(* IEC 61131-3 sources: SmartHomeNew/ (part 16) *)

(* ---- PRG_System.st ---- *)
PROGRAM PRG_System
VAR

// === SENSOR PROCESSING (SHADOW) ===
fbSensorCO : FB_Sensor_Analog_Processing;
fbCalibCO  : FB_Sensor_Calibration_Processor;
fbSensorMethane : FB_Sensor_Analog_Processing;
fbCalibMethane  : FB_Sensor_Calibration_Processor;
fbSmokeDetector : FB_Smoke_Detector;
L_CO_Processed : REAL;
L_CO_Calibrated : REAL;
L_Safety_Selector_i : INT;
L_Methane_Processed : REAL;
L_Methane_Calibrated : REAL;
L_Smoke_Detected : BOOL;

// === LIFETIME MANAGERS ===
fbLifetimePump : FB_Lifetime_Manager;
fbLifetimeFan  : FB_Lifetime_Manager;

    // === TREND WRITE CONTROL ===
    L_Trend_Write : BOOL;
    L_Trend_Write_Prev : BOOL;

    // === TREND → HISTORY BRIDGE ===
    L_Trend_Event : ST_History_Record;

    // === TREND SYSTEM (MVP) ===
    L_Trend_Logger : FB_Trend_Logger;
    L_Trend_Data : ST_Trend_Data;
    L_Trend_Adapter : FB_Trend_Adapter;
    L_Trend_Avg : REAL;
    L_Trend_Min : REAL;
    L_Trend_Max : REAL;
    L_Trend_Up : BOOL;
    L_Trend_Down : BOOL;
    L_Trend_Last_Write_MS : UDINT;
    L_Trend_Last_Written_Avg : REAL;
    L_Trend_Write_Allowed : BOOL;
    L_i : INT;
    L_Motion_Sensors_16 : ARRAY[1..16] OF BOOL;
    // --- ADAPTER LAYER ---
    L_Zone_Valves_8 : ARRAY[1..8] OF BOOL;
    L_Lighting_32   : ARRAY[1..32] OF BYTE;
    L_Lighting_Bool_32 : ARRAY[1..32] OF BOOL;
    L_FloorTemps_8  : ARRAY[1..8] OF REAL;
    fbCoreKernelObserver : FB_CoreKernel_Live_Observer;
    fbSystemHealth : FB_System_Health;
    fbRedundancy : FB_Redundancy_Manager;
    fbGateway : FB_Gateway_Interface;
    fbScenarioManager : FB_Scenario_Manager;
    fbScenarioGuard : FB_Scenario_Transition_Guard;
    fbSimulationManager : FB_Simulation_Manager;
    fbRuleEngine : FB_Rule_Engine;
    fbNVRAMManager : FB_NVRAM_Manager;

    fbBlackBox : FB_BlackBox_Recorder;
    fbAstroTimer : FB_Astro_Timer;
    fbAlarmManager : FB_Alarm_Manager;
    fbHistoryManager : FB_History_Manager;
    fbSafety : FB_Safety_Manager;
    fbStateManager : FB_State_Manager;
    fbWatchdog : FB_Watchdog;
    fbHMIInterface : FB_HMI_Interface;
    fbFaultLogger : FB_Fault_Logger;
    fbLogEvent : FB_LogEvent;

    L_Time_Diff : UDINT;
    L_Local_State : ST_System_State_Snapshot;
    L_Remote_State : ST_System_State_Snapshot;
    L_NVRAM_Cmd : BYTE;
    L_NVRAM_Offset : UDINT;
    L_NVRAM_Done : BOOL;
    L_NVRAM_Err : BOOL;
    L_NVRAM_ErrID : UDINT;
    L_BB_Record : ST_BlackBox_Record;
    L_BB_Freeze : BOOL;
    L_Scenario_Idx : INT;
        L_Last_Operator_Blocked : BOOL;
    L_Last_DHW_Heating_In_Service : BOOL;
    L_Last_DHW_Circ_In_Service : BOOL;
    L_Dangerous_Action_Armed : BOOL;
    L_Dangerous_Action_Deadline_MS : UDINT;
    L_Maintenance_Apply_Intent : BOOL;
    L_Last_System_Mode : E_System_Operating_Mode;
    L_Last_First_Fault_Type : INT;
    L_Last_First_Fault_Source : INT;
    L_Last_Root_Cause : E_System_Root_Cause;
    L_History_Event : ST_History_Record;
    L_History_Write_Event : BOOL;
    L_Last_Operator_Journal_Seq : UDINT;
    L_Last_Maintenance_Action_Code : UDINT;
    L_Last_Event_Code : UDINT;
    L_Last_Event_Value : REAL;
    L_Last_Event_Time_MS : UDINT;
    L_Gateway_Writes_Allowed : BOOL;
    L_Last_Policy_Event_Time_MS : UDINT;

    L_Scenario_Req_Operator : E_SCENARIO_TYPE;
    L_Scenario_Req_Gateway  : E_SCENARIO_TYPE;
    L_Scenario_Req_Rule     : E_SCENARIO_TYPE;
    L_Scenario_Req_Final    : E_SCENARIO_TYPE; // TRACE ONLY: arbitration result before policy
    L_Scenario_Intent       : E_SCENARIO_TYPE;
L_Scenario_Source       : E_SCENARIO_SOURCE;

L_IO_Fault_Prev : BOOL;
L_Watchdog_Fault_Prev : BOOL;
L_Comm_Fault_Prev : BOOL;
L_Sensor_Fault_Prev : BOOL;
L_Subsystem_Fault_Prev : BOOL;
L_Mode_Prev : E_System_Operating_Mode;
L_User_Access_Denied_Prev : BOOL;
L_Dangerous_Action_Request_Prev : BOOL;

    L_Persist_Buffer : ARRAY[0..4] OF BYTE;
    L_Last_Written_Persist_Buffer : ARRAY[0..4] OF BYTE;
    L_Persist_Buffer_Changed : BOOL;
    L_Last_Persist_Write_MS : UDINT;
    L_Recovery_Done : BOOL;
    L_Persist_Struct : ST_Persist;
END_VAR

// 0. Инициализация RETAIN переменных при первом запуске
IF NOT GVL_Retain.G_Initialized THEN
    FOR L_i := 0 TO GVL_CONSTANTS.C_MAX_PRESENCE_HISTORY - 1 DO
        GVL_Retain.G_Presence_History[L_i] := 0;
    END_FOR;

    GVL_Retain.G_History_Write_Idx := 1;
    GVL_Retain.G_History_Total_Events := 0;

    FOR L_i := 1 TO GVL_CONSTANTS.C_MAX_BOILERS DO
        GVL_Retain.G_Boiler_Accumulated_MS[L_i] := 0;
        GVL_Retain.G_Boiler_Work_Seconds[L_i] := 0;
    END_FOR;

    FOR L_i := 1 TO GVL_CONSTANTS.C_MAX_MANIFOLDS DO
        GVL_Retain.G_Valve_Test_Results[L_i] := FALSE;
    END_FOR;

    L_Local_State.Version := 0;
    L_Remote_State.Version := 0;

    GVL_Retain.G_Initialized := TRUE;

END_IF;

// === NVRAM RECOVERY (ONCE AFTER BOOT) ===
IF NOT L_Recovery_Done THEN
    IF GVL_PERSISTENT.P_Valid THEN
        GVL_STATE.G_Safety_Gas_Latched := GVL_PERSISTENT.P_Safety_Gas_Latched;
        GVL_STATE.G_Safety_Smoke_Latched := GVL_PERSISTENT.P_Safety_Smoke_Latched;
        GVL_STATE.G_Safety_Leak_Latched := GVL_PERSISTENT.P_Safety_Leak_Latched;
        GVL_STATE.G_System_Mode := GVL_PERSISTENT.P_System_Mode;
    END_IF;

    L_Recovery_Done := TRUE;
END_IF;

// NVRAM CONTROLLED WRITE ENABLED (step 8B)

// 1. Обновление системного времени
GVL_STATUS.G_System_Time_MS := TIME_TO_UDINT(TIME());
L_Time_Diff := (SEL(GVL_STATUS.G_System_Time_MS >= GVL_STATUS.G_Last_System_Time_MS, GVL_STATUS.G_System_Time_MS - GVL_STATUS.G_Last_System_Time_MS, (4294967295 - GVL_STATUS.G_Last_System_Time_MS) + GVL_STATUS.G_System_Time_MS + 1));
GVL_STATUS.G_Time_Of_Day_MS := (GVL_STATUS.G_Time_Of_Day_MS + L_Time_Diff) MOD 86400000;

IF GVL_STATUS.G_Time_Of_Day_MS < L_Time_Diff THEN
    GVL_STATUS.G_Current_Day := (GVL_STATUS.G_Current_Day MOD 7) + 1;
    GVL_STATUS.G_Day_Of_Year := (GVL_STATUS.G_Day_Of_Year MOD 365) + 1;
END_IF;

GVL_STATUS.G_Last_System_Time_MS := GVL_STATUS.G_System_Time_MS;
GVL_STATUS.G_Current_TOD := UDINT_TO_TOD(GVL_STATUS.G_Time_Of_Day_MS);

// Формирование локального состояния для репликации
L_Local_State.System_Time_MS := GVL_STATUS.G_System_Time_MS;
L_Local_State.Current_Scenario := GVL_STATUS.G_Current_Scenario;
L_Local_State.Security_Armed := GVL_ALARM.G_Security_Armed;
L_Local_State.Active_Alarms := GVL_ALARM.G_Active_Alarm_Count;
L_Local_State.Zone_Valves := GVL_STATE.G_Zone_Valves;
L_Local_State.Manifold_Pumps := GVL_STATE.G_Manifold_Pumps;
L_Local_State.Lighting_States := GVL_STATE.G_Lighting_Levels;
L_Local_State.Blinds_Positions := GVL_STATE.G_Blinds_Positions;
L_Local_State.Socket_States := GVL_STATE.G_Socket_States;
L_Local_State.Gas_Valve_Closed := GVL_COMMAND.G_Gas_Valve_Close;
L_Local_State.Water_Valves_Closed := GVL_COMMAND.G_Close_Valve_36;
L_Local_State.Version := L_Local_State.Version + 1;

// 2. Определение роли ПЛК (Active/Standby)
fbRedundancy(
    VI_System_Time_MS := GVL_STATUS.G_System_Time_MS,
    VI_Local_PLC_ID := GVL_STATUS.G_PLC_ID,
    VI_Remote_Pulse := GVL_IO.DI_Partner_Pulse,
    VI_Remote_Is_Active := GVL_IO.DI_Partner_Active,
    VI_Gateway_Ping_OK := GVL_GATEWAY.G_Gateway_Ping_OK,
    VI_Local_State := L_Local_State,
    VI_Remote_State := L_Remote_State
);
GVL_STATUS.G_Is_Active_PLC := (fbRedundancy.VO_Local_Role = E_PLC_ROLE.ROLE_ACTIVE);
GVL_IO.DO_Heartbeat_Pulse := fbRedundancy.VO_Local_Pulse;
GVL_IO.DO_Active_Status := GVL_STATUS.G_Is_Active_PLC;

// 3. Синхронизация состояния (применение полученного состояния)
IF fbRedundancy.VO_State_Updated THEN
    GVL_STATUS.G_Current_Scenario := fbRedundancy.VO_Synced_State.Current_Scenario;
    GVL_ALARM.G_Security_Armed := fbRedundancy.VO_Synced_State.Security_Armed;
    GVL_STATE.G_Zone_Valves := fbRedundancy.VO_Synced_State.Zone_Valves;
    GVL_STATE.G_Manifold_Pumps := fbRedundancy.VO_Synced_State.Manifold_Pumps;
    GVL_STATE.G_Lighting_Levels := fbRedundancy.VO_Synced_State.Lighting_States;
    GVL_STATE.G_Blinds_Positions := fbRedundancy.VO_Synced_State.Blinds_Positions;
    GVL_STATE.G_Socket_States := fbRedundancy.VO_Synced_State.Socket_States;
    GVL_COMMAND.G_Gas_Valve_Close := fbRedundancy.VO_Synced_State.Gas_Valve_Closed;
    GVL_COMMAND.G_Close_Valve_36 := fbRedundancy.VO_Synced_State.Water_Valves_Closed;
    L_Local_State.Version := fbRedundancy.VO_Synced_State.Version;
END_IF;

fbSafety(
    VI_Gas_Alarm := GVL_STATE.G_Safety_Gas_Alarm,
    VI_Leak_Alarm := GVL_STATE.G_Safety_Leak_Alarm,
    VI_Smoke_Alarm := GVL_STATE.G_Safety_Smoke_Alarm,
    VI_Reset := GVL_COMMAND.G_Reset_Errors,
    VO_Gas_Latched => GVL_STATE.G_Safety_Gas_Latched,
    VO_Leak_Latched => GVL_STATE.G_Safety_Leak_Latched,
    VO_Smoke_Latched => GVL_STATE.G_Safety_Smoke_Latched,
    VO_Emergency_Stop => GVL_STATE.G_Safety_Emergency_Stop
);

// 3.4. Агрегация состояния anti-freeze hardware
GVL_STATE.G_Freeze_Hardware_Degraded := GVL_STATUS.G_Diagnostics.Backup_Pump_Fault OR GVL_STATUS.G_Diagnostics.Electric_Heater_Fault;
GVL_STATE.G_Freeze_Hardware_Failed := GVL_STATUS.G_Diagnostics.Backup_Pump_Fault AND GVL_STATUS.G_Diagnostics.Electric_Heater_Fault;

// 3.6. Health manager: новая интеграция safety + diagnostics + watchdog
fbWatchdog(
    VI_System_Time_MS := GVL_STATUS.G_System_Time_MS
);

fbSystemHealth(
    VI_Smoke_Detected := GVL_HEALTH_BRIDGE.G_Smoke_Detected OR GVL_STATE.G_Safety_Smoke_Latched,
    VI_Gas_Detected := GVL_HEALTH_BRIDGE.G_Gas_Detected OR GVL_STATE.G_Safety_Gas_Latched,
    VI_CO_Warning_Level := GVL_HEALTH_BRIDGE.G_CO_Warning_Level,
    VI_CO_Alarm_Level := GVL_HEALTH_BRIDGE.G_CO_Alarm_Level,
    VI_Leak_Detected := GVL_HEALTH_BRIDGE.G_Leak_Detected OR GVL_STATE.G_Safety_Leak_Latched,
    VI_Sensor_Fault := GVL_STATE.G_Heating_Sensor_Fault OR GVL_STATE.G_DHW_Sensor_Fault,
    VI_IO_Offline := GVL_STATE.G_Heating_IO_Fault OR GVL_STATE.G_DHW_IO_Fault OR GVL_STATE.G_Ventilation_IO_Fault OR GVL_STATE.G_Lighting_IO_Fault,
    VI_Comm_Fault := GVL_STATE.G_Access_Comm_Fault,
    VI_Watchdog_Fault := fbWatchdog.VO_Watchdog_Fault,
    VI_Subsystem_Fault := GVL_STATE.G_Heating_Subsystem_Degraded OR GVL_STATE.G_DHW_Subsystem_Degraded OR GVL_STATE.G_Ventilation_Subsystem_Degraded
);

// 3.6. State manager: агрегированная логика режима работы
fbStateManager(
    VI_System_Severity := fbSystemHealth.VO_System_Severity,
    VI_Root_Cause := fbSystemHealth.VO_Root_Cause,
    VI_Freeze_Risk := GVL_STATE.G_Safety_Freeze_Risk
);

fbHMIInterface(
    VI_Severity := fbSystemHealth.VO_System_Severity,
    VI_RootCause := fbSystemHealth.VO_Root_Cause,
    VI_Status_Msg := fbStateManager.VO_Status_Msg
);

fbFaultLogger(
    VI_Severity := fbSystemHealth.VO_System_Severity,
    VI_RootCause := fbSystemHealth.VO_Root_Cause,
    VI_Time_MS := GVL_STATUS.G_System_Time_MS
);

// publish integrated outputs
GVL_STATUS.G_System_Mode_Msg := fbStateManager.VO_Status_Msg;

// === DIAGNOSTIC FLAGS (export) ===
GVL_STATUS.G_Diagnostics.Sensor_Fault :=
    GVL_STATE.G_Heating_Sensor_Fault OR
    GVL_STATE.G_DHW_Sensor_Fault;

GVL_STATUS.G_Diagnostics.IO_Offline :=
    GVL_STATE.G_Heating_IO_Fault OR
    GVL_STATE.G_DHW_IO_Fault OR
    GVL_STATE.G_Ventilation_IO_Fault OR
    GVL_STATE.G_Lighting_IO_Fault;

GVL_STATUS.G_Diagnostics.Subsystem_Degraded :=
    GVL_STATE.G_Heating_Subsystem_Degraded OR
    GVL_STATE.G_DHW_Subsystem_Degraded OR
    GVL_STATE.G_Ventilation_Subsystem_Degraded;

GVL_GATEWAY.G_Gateway_HMI_Status_Message := fbHMIInterface.VO_HMI_Status_Text;
IF fbFaultLogger.VO_Last_Event_Text <> '' THEN
    GVL_HEALTH_BRIDGE.G_Last_Fault_Event_Text := fbFaultLogger.VO_Last_Event_Text;
END_IF;

// 3.7. Применение вычисленного режима системы
GVL_STATE.G_System_Mode := fbStateManager.VO_System_Mode;

CASE GVL_STATE.G_System_Mode OF
    E_System_Operating_Mode.MODE_SAFE_STOP:
        GVL_STATE.G_System_Mode_Text := 'SAFE_STOP';

    E_System_Operating_Mode.MODE_FREEZE_PROTECTION:
        GVL_STATE.G_System_Mode_Text := 'FREEZE_PROTECTION';

    E_System_Operating_Mode.MODE_DEGRADED:
        GVL_STATE.G_System_Mode_Text := 'DEGRADED';

    ELSE
        GVL_STATE.G_System_Mode_Text := 'NORMAL';
END_CASE;

CASE fbSystemHealth.VO_Root_Cause OF
    E_System_Root_Cause.ROOT_FIRE:
        GVL_STATUS.G_System_Mode_Cause := 'Пожар/дым';
    E_System_Root_Cause.ROOT_GAS_LEAK:
        GVL_STATUS.G_System_Mode_Cause := 'Утечка газа';
    E_System_Root_Cause.ROOT_CO_CRITICAL:
        GVL_STATUS.G_System_Mode_Cause := 'Критический CO';
    E_System_Root_Cause.ROOT_CO_WARNING:
        GVL_STATUS.G_System_Mode_Cause := 'Повышенный CO';
    E_System_Root_Cause.ROOT_WATER_LEAK:
        GVL_STATUS.G_System_Mode_Cause := 'Протечка воды';
    E_System_Root_Cause.ROOT_WATCHDOG_FAULT:
        GVL_STATUS.G_System_Mode_Cause := 'Ошибка watchdog';
    E_System_Root_Cause.ROOT_IO_OFFLINE:
        GVL_STATUS.G_System_Mode_Cause := 'Недоступен модуль IO';
    E_System_Root_Cause.ROOT_COMM_FAULT:
        GVL_STATUS.G_System_Mode_Cause := 'Ошибка связи';
    E_System_Root_Cause.ROOT_SENSOR_FAULT:
        GVL_STATUS.G_System_Mode_Cause := 'Ошибка датчика';
    E_System_Root_Cause.ROOT_SUBSYSTEM_FAULT:
        GVL_STATUS.G_System_Mode_Cause := 'Ошибка подсистемы';
    ELSE
        GVL_STATUS.G_System_Mode_Cause := 'Аварийные режимы отсутствуют';
END_CASE;

// final status text comes from State_Manager
GVL_STATUS.G_System_Mode_Msg := fbStateManager.VO_Status_Msg;

// 3.6a. Расчёт направленной эвакуации
FOR L_i := 1 TO 32 DO
    GVL_STATE.G_Evac_Guidance[L_i] := 0;

    IF GVL_STATE.G_Evac_Hazard_Zone[L_i] THEN
        GVL_STATE.G_Evac_Guidance[L_i] := -1;
    END_IF;

    IF GVL_CONFIG.G_Evac_Exit_Zones[L_i] AND NOT GVL_STATE.G_Evac_Hazard_Zone[L_i] THEN
        GVL_STATE.G_Evac_Guidance[L_i] := 1;
    END_IF;
END_FOR;

// 3.5a. Вычисление человекочитаемых имён зон эвакуации для HMI
GVL_STATUS.G_Evac_Target_Zone_Name := '';
GVL_STATUS.G_Evac_Hazard_Zone_Name := '';

FOR L_i := 1 TO 32 DO
    IF (GVL_STATUS.G_Evac_Hazard_Zone_Name = '') AND GVL_STATE.G_Evac_Hazard_Zone[L_i] THEN
        GVL_STATUS.G_Evac_Hazard_Zone_Name := GVL_CONFIG.G_Evac_Zone_Names[L_i];
        IF GVL_STATUS.G_Evac_Hazard_Zone_Name = '' THEN
            GVL_STATUS.G_Evac_Hazard_Zone_Name := CONCAT('Zone ', INT_TO_STRING(L_i));
        END_IF;
    END_IF;

    IF (GVL_STATUS.G_Evac_Target_Zone_Name = '') AND (GVL_STATE.G_Evac_Guidance[L_i] = 1) THEN
        GVL_STATUS.G_Evac_Target_Zone_Name := GVL_CONFIG.G_Evac_Zone_Names[L_i];
        IF GVL_STATUS.G_Evac_Target_Zone_Name = '' THEN
            GVL_STATUS.G_Evac_Target_Zone_Name := CONCAT('Zone ', INT_TO_STRING(L_i));
        END_IF;
    END_IF;
END_FOR;

// 3.6. Активация световой эвакуации
IF GVL_STATE.G_System_Mode = E_System_Operating_Mode.MODE_SAFE_STOP AND GVL_STATE.G_Safety_Smoke_Latched THEN
    GVL_STATE.G_Evacuation_Lighting_Active := TRUE;
ELSE
    GVL_STATE.G_Evacuation_Lighting_Active := FALSE;
END_IF;

// 4. Астрономический таймер
fbAstroTimer(
    VI_System_Time_MS := GVL_STATUS.G_System_Time_MS,
    VI_Latitude := 55.75,
    VI_Longitude := 37.61,
    VI_Day_Of_Year := GVL_STATUS.G_Day_Of_Year,
    VO_Is_Night => GVL_STATUS.G_Is_Night
);

// 5. Управление сценариями
// Scenario request (direct + early operator gate)
IF GVL_STATE.G_System_Mode = E_System_Operating_Mode.MODE_NORMAL THEN
    L_Scenario_Req_Operator := GVL_COMMAND.G_Scenario_Request_Operator;
ELSE
    L_Scenario_Req_Operator := E_SCENARIO_TYPE.SCENARIO_NONE;
END_IF;
L_Scenario_Req_Gateway := 0;
L_Scenario_Req_Rule := 0;

// Синхронизируем request с фактически активным сценарием

L_Scenario_Idx := TO_INT(GVL_STATUS.G_Current_Scenario);
IF L_Scenario_Idx < 0 OR L_Scenario_Idx > 7 THEN
    L_Scenario_Idx := 0;
END_IF;

// 6. Симуляция присутствия
fbSimulationManager(
    VI_System_Time_MS := GVL_STATUS.G_System_Time_MS,
    VI_IsActivePLC := GVL_STATUS.G_Is_Active_PLC AND (GVL_STATE.G_System_Mode = E_System_Operating_Mode.MODE_NORMAL),
    VI_Scenario := GVL_STATUS.G_Current_Scenario,
    VI_Config := GVL_CONFIG.G_HMI_Scenario_Configs[L_Scenario_Idx],
    VO_Sim_Lights => GVL_STATE.G_Sim_Lights,
    VO_Sim_Active => GVL_STATUS.G_Sim_Active
);

// 6.5. Пользовательские правила (Rule Engine)
fbRuleEngine(
    VI_System_Time_MS := GVL_STATUS.G_System_Time_MS,
    VI_IsActivePLC := GVL_STATUS.G_Is_Active_PLC,
    VI_Rules := GVL_CONFIG.G_HMI_User_Rules,
    VI_Indoor_Temps := GVL_STATE.G_Room_Temps,
    VI_Floor_Temps := L_FloorTemps_8,
    VI_Humidities := GVL_STATE.G_Room_Hum,
    VI_CO2_Levels := GVL_STATE.G_Room_CO2,
    VI_Motion_Sensors := L_Motion_Sensors_16,
    VI_Door_Sensors := GVL_STATE.G_Door_Sensors,
    VI_Window_Sensors := GVL_STATE.G_Window_Sensors,
    VI_Water_Sensors := GVL_STATE.G_Water_Sensors,
    VI_Smoke_Sensors := GVL_STATE.G_Smoke_Sensors,
    VI_Methane_Sensors := GVL_STATE.G_Methane_Sensors,
    VI_CO_Sensors := GVL_STATE.G_CO_Sensors,
    VI_Security_Armed := GVL_ALARM.G_Security_Armed,
    VI_Current_Time := GVL_STATUS.G_Current_TOD,
    VI_Day_Of_Week := TO_INT(GVL_STATUS.G_Current_Day),
    VO_Actions => GVL_STATE.G_Rule_Actions
);

FOR L_i := 1 TO GVL_CONSTANTS.C_MAX_RULES DO
    IF GVL_STATE.G_Rule_Actions[L_i].Active AND GVL_STATE.G_Rule_Actions[L_i].Action_Type = E_Rule_Action_Type.ACTION_ACTIVATE_SCENARIO THEN
        L_Scenario_Req_Rule := TO_BYTE(GVL_STATE.G_Rule_Actions[L_i].Value);
    END_IF;
END_FOR;

// 8.5 Менеджер тревог (Сбор всех аварий)
fbAlarmManager(
    VI_System_Time_MS := GVL_STATUS.G_System_Time_MS,
    VI_IsActivePLC := GVL_STATUS.G_Is_Active_PLC,
    VI_Gas_Alarm := GVL_ALARM.G_Gas_Alarm_Active,
    VI_Fire_Alarm := GVL_ALARM.G_Fire_Alarm_Active,
    VI_Flood_Alarm := GVL_ALARM.G_Flood_Alarm_Active,
    VI_Security_Alarm := GVL_ALARM.G_Security_Alarm,
    VI_First_Fault_Active := fbSystemHealth.VO_First_Fault_Active,
    VI_First_Fault_Type := fbSystemHealth.VO_First_Fault_Type,
    VI_First_Fault_Source := fbSystemHealth.VO_First_Fault_Source,
    VI_Boiler_Errors := GVL_STATE.G_Boiler_Error,
    VI_Security_Msg := GVL_STATUS.G_Security_Status_Msg,
    VI_Acknowledge_All := GVL_CONFIG.G_HMI_Ack_Alarms OR GVL_COMMAND.G_Reset_Errors,
    VI_Mute_Siren := GVL_CONFIG.G_HMI_Mute_Alarm,
    VIO_Next_Alarm_ID := GVL_ALARM.G_Next_Alarm_ID,
    VO_Global_Critical => GVL_ALARM.G_Global_Critical,
    VO_Global_Warning => GVL_ALARM.G_Global_Warning,
    VO_Siren_Active => GVL_ALARM.G_Global_Siren,
    VO_Active_Count => GVL_ALARM.G_Active_Alarm_Count,
    VO_Unacked_Count => GVL_ALARM.G_Unacked_Alarm_Count,
    VO_Event_Pulse => GVL_STATUS.G_Diagnostics.Alarm_Event_Pulse,
    VO_Event_Code => GVL_STATUS.G_Diagnostics.Alarm_Event_Code,
    VO_Event_Value => GVL_STATUS.G_Diagnostics.Alarm_Event_Value,
    VO_Alarm_List => GVL_ALARM.G_Alarm_List
);

// Command arbitration: OPERATOR > GATEWAY
L_Gateway_Writes_Allowed :=
    NOT GVL_STATUS.G_Diagnostics.Dangerous_Action_Pending_Confirm AND
    NOT GVL_STATUS.G_Diagnostics.Operator_Action_Blocked AND
    NOT GVL_STATUS.G_Diagnostics.User_Access_Denied;

// 13. Интерфейс шлюза (Modbus TCP)
fbGateway(
    VI_System_Time_MS := GVL_STATUS.G_System_Time_MS,
    VI_Local_PLC_Role := SEL(GVL_STATUS.G_Is_Active_PLC, E_PLC_ROLE.ROLE_STANDBY, E_PLC_ROLE.ROLE_ACTIVE),
    VI_Incoming_Command := GVL_GATEWAY.G_Gateway_Command,
    VI_Command_Received := GVL_GATEWAY.G_Gateway_Command_Received,
    VI_FloorHeating_Temps := L_FloorTemps_8,
    VI_Room_Temps := GVL_STATE.G_Room_Temps,
    VI_Zone_Valve_States := L_Zone_Valves_8,
    VI_Manifold_Pressures := GVL_STATE.G_Manifold_Pressures,
    VI_Manifold_Pump_States := GVL_STATE.G_Manifold_Pumps,
    VI_Outdoor_Temp := GVL_STATE.G_Outdoor_Temp,
    VI_Security_Armed := GVL_ALARM.G_Security_Armed,
    VI_Flood_Alarm_Active := GVL_ALARM.G_Flood_Alarm_Active,
    VI_Gas_Alarm_Active := GVL_ALARM.G_Gas_Alarm_Active,
    VI_Fire_Alarm_Active := GVL_ALARM.G_Fire_Alarm_Active,
    VI_Methane_Concentration := GVL_STATE.G_Methane_Sensors[1],
    VI_Lighting_Base_Levels := L_Lighting_32,
    VI_Socket_States := GVL_STATE.G_Socket_States,
    VI_Blinds_Positions := GVL_STATE.G_Blinds_Positions,
    VI_Active_Scenario := GVL_STATUS.G_Current_Scenario,
    VI_Send_2FA_Req := GVL_COMMAND.G_Send_2FA_Req,
    VI_2FA_Code := GVL_COMMAND.G_2FA_Code_Out,
    VI_Allowed_IPs := GVL_CONFIG.G_Allowed_IPs,
    VO_Telegram_Msg => GVL_GATEWAY.G_Gateway_Telegram_Msg,
    VO_Send_Telegram => GVL_GATEWAY.G_Gateway_Send_Telegram,
    VO_HMI_Status_Message => GVL_GATEWAY.G_Gateway_HMI_Status_Message,

    VO_Data_Ready => GVL_GATEWAY.G_Gateway_Data_Ready,
    VO_Modbus_Registers => GVL_GATEWAY.G_Gateway_Modbus_Registers,
    VO_Arm_Req => GVL_COMMAND.G_Arm_Req,
    VO_Disarm_Req => GVL_COMMAND.G_Disarm_Req,
    VO_PIN_Code => GVL_COMMAND.G_PIN_Code,
    VO_RFID_Tag => GVL_COMMAND.G_RFID_Tag,
    VO_2FA_Code_In => GVL_COMMAND.G_2FA_Code_In,
    VO_Lighting_Override => GVL_COMMAND.G_Lighting_Override,
    VO_Blinds_Override => GVL_COMMAND.G_Blinds_Override,
    VO_Socket_Override => GVL_COMMAND.G_Socket_Override,
    VO_Reset_Errors_Req => GVL_COMMAND.G_Reset_Errors
);

IF L_Gateway_Writes_Allowed AND
   fbGateway.VO_Set_Scenario_Req AND
   ((GVL_STATE.G_System_Mode = E_System_Operating_Mode.MODE_NORMAL) OR
    (GVL_STATE.G_System_Mode = E_System_Operating_Mode.MODE_DEGRADED)) THEN
    L_Scenario_Req_Gateway := fbGateway.VO_Target_Scenario;
END_IF;

IF L_Gateway_Writes_Allowed AND
   fbGateway.VO_Set_Temp_Req AND
   (GVL_STATE.G_System_Mode = E_System_Operating_Mode.MODE_NORMAL) THEN
    GVL_CONFIG.G_HMI_FloorHeating_Configs[fbGateway.VO_Target_Zone].design_temp := fbGateway.VO_Target_Temp;
END_IF;

IF L_Gateway_Writes_Allowed AND
   fbGateway.VO_Set_Vent_Req AND
   (GVL_STATE.G_System_Mode = E_System_Operating_Mode.MODE_NORMAL) THEN
    GVL_CONFIG.G_HMI_Vent_Global_Config.default_supply_speed := fbGateway.VO_Target_Vent_Speed;
END_IF;

IF L_Gateway_Writes_Allowed AND
   fbGateway.VO_Set_Config_Req AND
   (GVL_STATE.G_System_Mode = E_System_Operating_Mode.MODE_NORMAL) THEN
    GVL_CONFIG.G_HMI_Apply_Settings := TRUE;
END_IF;

IF L_Gateway_Writes_Allowed AND
   fbGateway.VO_Sync_Time_Req AND
   (GVL_STATE.G_System_Mode = E_System_Operating_Mode.MODE_NORMAL) THEN
    GVL_STATUS.G_Time_Of_Day_MS := fbGateway.VO_New_Time_MS;
END_IF;

// === SCENARIO REQUEST VALIDATION ===
// Normalize invalid values to NONE to avoid corrupt inputs.
// Actual enum range in E_SCENARIO_TYPE is 0..7.
IF TO_USINT(L_Scenario_Req_Operator) > 7 THEN
    L_Scenario_Req_Operator := E_SCENARIO_TYPE.SCENARIO_NONE;
END_IF;

IF TO_USINT(L_Scenario_Req_Gateway) > 7 THEN
    L_Scenario_Req_Gateway := E_SCENARIO_TYPE.SCENARIO_NONE;
END_IF;

IF TO_USINT(L_Scenario_Req_Rule) > 7 THEN
    L_Scenario_Req_Rule := E_SCENARIO_TYPE.SCENARIO_NONE;
END_IF;

// ================= COMMAND GATE (FINAL) =================
IF GVL_STATE.G_System_Mode = E_System_Operating_Mode.MODE_SAFE_STOP THEN

    // Блокируем ВСЕ опасные команды после Gateway
    GVL_COMMAND.G_Scenario_Request_Operator := 0;

    FOR L_i := 1 TO 32 DO
        GVL_COMMAND.G_Lighting_Override[L_i] := BYTE#0;
        GVL_COMMAND.G_Blinds_Override[L_i] := BYTE#0;
        GVL_COMMAND.G_Socket_Override[L_i] := FALSE;
    END_FOR;

    // НЕ блокируем:
    // G_Reset_Errors
    // acknowledge / безопасность

END_IF;
// =======================================================

// === SCENARIO PRIORITY RESOLUTION ===
// Produces L_Scenario_Req_Final (TRACE ONLY, not executed directly)
IF GVL_STATE.G_System_Mode = E_System_Operating_Mode.MODE_SAFE_STOP THEN
    L_Scenario_Req_Final := 0;
    L_Scenario_Source := SRC_SAFETY;
ELSIF L_Scenario_Req_Operator <> 0 THEN
    L_Scenario_Req_Final := L_Scenario_Req_Operator;
    L_Scenario_Source := SRC_OPERATOR;
ELSIF L_Scenario_Req_Gateway <> 0 THEN
    L_Scenario_Req_Final := L_Scenario_Req_Gateway;
    L_Scenario_Source := SRC_GATEWAY;
ELSIF L_Scenario_Req_Rule <> 0 THEN
    L_Scenario_Req_Final := L_Scenario_Req_Rule;
    L_Scenario_Source := SRC_RULE;
ELSE
    L_Scenario_Req_Final := GVL_STATUS.G_Current_Scenario;
    L_Scenario_Source := SRC_NONE;
END_IF;

L_Scenario_Intent := L_Scenario_Req_Final;

// === FAIL-SAFE SCENARIO CLAMP ===
CASE GVL_STATE.G_System_Mode OF
    E_System_Operating_Mode.MODE_SAFE_STOP:
        L_Scenario_Intent := E_SCENARIO_TYPE.SCENARIO_NONE;

    E_System_Operating_Mode.MODE_FREEZE_PROTECTION:
        L_Scenario_Intent := E_SCENARIO_TYPE.SCENARIO_NONE;

    E_System_Operating_Mode.MODE_DEGRADED:
        CASE L_Scenario_Intent OF
            E_SCENARIO_TYPE.SCENARIO_NONE,
            E_SCENARIO_TYPE.SCENARIO_PRESENCE,
            E_SCENARIO_TYPE.SCENARIO_AWAY,
            E_SCENARIO_TYPE.SCENARIO_SLEEP:
                ; // allowed in degraded
        ELSE
            L_Scenario_Intent := E_SCENARIO_TYPE.SCENARIO_NONE;
        END_CASE;
END_CASE;

// === CONTEXT FAIL-SAFE AUTOMATION ===
// If security is armed and no explicit source is requesting another scenario,
// force safe occupancy context to AWAY while system remains in MODE_NORMAL.
IF GVL_STATE.G_System_Mode = E_System_Operating_Mode.MODE_NORMAL THEN
    IF GVL_ALARM.G_Security_Armed AND
       (L_Scenario_Req_Operator = E_SCENARIO_TYPE.SCENARIO_NONE) AND
       (L_Scenario_Req_Gateway = E_SCENARIO_TYPE.SCENARIO_NONE) AND
       (L_Scenario_Req_Rule = E_SCENARIO_TYPE.SCENARIO_NONE) AND
       (L_Scenario_Intent <> E_SCENARIO_TYPE.SCENARIO_AWAY) THEN

        IF L_Scenario_Intent <> E_SCENARIO_TYPE.SCENARIO_AWAY THEN
            L_Scenario_Intent := E_SCENARIO_TYPE.SCENARIO_AWAY;
            L_Scenario_Source := SRC_POLICY;

            IF (L_Last_Policy_Event_Time_MS = 0) OR
               ((GVL_STATUS.G_System_Time_MS - L_Last_Policy_Event_Time_MS) >= 5000) THEN
                fbLogEvent(
                    VI_Event_Type := 5,
                    VI_Timestamp := GVL_STATUS.G_System_Time_MS,
                    VI_Param1 := TO_UDINT(L_Scenario_Source),
                    VI_Param2 := TO_UDINT(E_SCENARIO_TYPE.SCENARIO_AWAY)
                );
                L_Last_Policy_Event_Time_MS := GVL_STATUS.G_System_Time_MS;
            END_IF;
        END_IF;
    END_IF;
END_IF;

// === DEGRADED-AWARE SCENARIO ADAPTATION ===
// Soft adaptation in degraded mode: keep explicit requests intact,
// but if no source is requesting a scenario, move behavior to a safer baseline.
IF GVL_STATE.G_System_Mode = E_System_Operating_Mode.MODE_DEGRADED THEN
    IF (L_Scenario_Req_Operator = E_SCENARIO_TYPE.SCENARIO_NONE) AND
       (L_Scenario_Req_Gateway = E_SCENARIO_TYPE.SCENARIO_NONE) AND
       (L_Scenario_Req_Rule = E_SCENARIO_TYPE.SCENARIO_NONE) THEN

        IF GVL_ALARM.G_Security_Armed THEN
            IF L_Scenario_Intent <> E_SCENARIO_TYPE.SCENARIO_AWAY THEN
                L_Scenario_Intent := E_SCENARIO_TYPE.SCENARIO_AWAY;
                L_Scenario_Source := SRC_POLICY;

                IF (L_Last_Policy_Event_Time_MS = 0) OR
                   ((GVL_STATUS.G_System_Time_MS - L_Last_Policy_Event_Time_MS) >= 5000) THEN
                    fbLogEvent(
                        VI_Event_Type := 6,
                        VI_Timestamp := GVL_STATUS.G_System_Time_MS,
                        VI_Param1 := TO_UDINT(L_Scenario_Source),
                        VI_Param2 := TO_UDINT(E_SCENARIO_TYPE.SCENARIO_AWAY)
                    );
                    L_Last_Policy_Event_Time_MS := GVL_STATUS.G_System_Time_MS;
                END_IF;
            END_IF;

        ELSIF L_Scenario_Intent = E_SCENARIO_TYPE.SCENARIO_PRESENCE THEN
            IF L_Scenario_Intent <> E_SCENARIO_TYPE.SCENARIO_SLEEP THEN
                L_Scenario_Intent := E_SCENARIO_TYPE.SCENARIO_SLEEP;
                L_Scenario_Source := SRC_POLICY;

                IF (L_Last_Policy_Event_Time_MS = 0) OR
                   ((GVL_STATUS.G_System_Time_MS - L_Last_Policy_Event_Time_MS) >= 5000) THEN
                    fbLogEvent(
                        VI_Event_Type := 7,
                        VI_Timestamp := GVL_STATUS.G_System_Time_MS,
                        VI_Param1 := TO_UDINT(L_Scenario_Source),
                        VI_Param2 := TO_UDINT(E_SCENARIO_TYPE.SCENARIO_SLEEP)
                    );
                    L_Last_Policy_Event_Time_MS := GVL_STATUS.G_System_Time_MS;
                END_IF;
            END_IF;
        END_IF;
    END_IF;
END_IF;

fbScenarioGuard(
    VI_Current_Scenario := GVL_STATUS.G_Current_Scenario,
    VI_Target_Scenario := L_Scenario_Intent
);

IF NOT fbScenarioGuard.VO_Transition_Allowed THEN
    GVL_GATEWAY.G_Gateway_HMI_Status_Message := CONCAT('Scenario guard: ', fbScenarioGuard.VO_Reason);
    L_Scenario_Intent := GVL_STATUS.G_Current_Scenario;
END_IF;

fbScenarioManager(
    VI_System_Time_MS := GVL_STATUS.G_System_Time_MS,
    VI_Activate_Request := L_Scenario_Intent,
    VI_IsActivePLC := GVL_STATUS.G_Is_Active_PLC,
    VI_System_Mode := GVL_STATE.G_System_Mode,
    VO_Current_Scenario => GVL_STATUS.G_Current_Scenario
);

// 14. Менеджер NVRAM
// Pack persistent snapshot into compact byte buffer for controlled NVRAM mirroring
L_Persist_Buffer[0] := TO_BYTE(TO_INT(L_Persist_Struct.System_Mode));
IF L_Persist_Struct.Safety_Gas_Latched THEN
    L_Persist_Buffer[1] := BYTE#1;
ELSE
    L_Persist_Buffer[1] := BYTE#0;
END_IF;
IF L_Persist_Struct.Safety_Smoke_Latched THEN
    L_Persist_Buffer[2] := BYTE#1;
ELSE
    L_Persist_Buffer[2] := BYTE#0;
END_IF;
IF L_Persist_Struct.Safety_Leak_Latched THEN
    L_Persist_Buffer[3] := BYTE#1;
ELSE
    L_Persist_Buffer[3] := BYTE#0;
END_IF;
IF L_Persist_Struct.DHW_Heating_Pump THEN
    L_Persist_Buffer[4] := BYTE#1;
ELSE
    L_Persist_Buffer[4] := BYTE#0;
END_IF;

L_Persist_Buffer_Changed :=
    (L_Persist_Buffer[0] <> L_Last_Written_Persist_Buffer[0]) OR
    (L_Persist_Buffer[1] <> L_Last_Written_Persist_Buffer[1]) OR
    (L_Persist_Buffer[2] <> L_Last_Written_Persist_Buffer[2]) OR
    (L_Persist_Buffer[3] <> L_Last_Written_Persist_Buffer[3]) OR
    (L_Persist_Buffer[4] <> L_Last_Written_Persist_Buffer[4]);

L_NVRAM_Cmd := 0;
L_NVRAM_Offset := 0;

IF GVL_CONFIG.G_HMI_Apply_Settings THEN
    // explicit config apply may request a controlled write
    L_NVRAM_Cmd := 1;
    GVL_CONFIG.G_HMI_Apply_Settings := FALSE;

ELSIF L_Persist_Buffer_Changed THEN
    // controlled write: no more often than once per 60 seconds
    IF (L_Last_Persist_Write_MS = 0) OR
       ((GVL_STATUS.G_System_Time_MS - L_Last_Persist_Write_MS) >= 60000) THEN
        L_NVRAM_Cmd := 1;
    END_IF;
END_IF;

fbNVRAMManager(
    VI_Command := L_NVRAM_Cmd,
    VI_Offset := L_NVRAM_Offset,
    VI_DataRef := L_Persist_Buffer[0],
    VI_DataSize := 5,
    VI_System_Time_MS := GVL_STATUS.G_System_Time_MS,
    VI_Operator_ID := 'SYSTEM',
    VI_IsActivePLC := GVL_STATUS.G_Is_Active_PLC,
    VI_TwoPersonConfirmation := FALSE,
    VO_Done => L_NVRAM_Done,
    VO_Error => L_NVRAM_Err,
    VO_ErrorID => L_NVRAM_ErrID
);

IF (L_NVRAM_Cmd = 1) AND L_NVRAM_Done AND NOT L_NVRAM_Err THEN
    L_Last_Written_Persist_Buffer[0] := L_Persist_Buffer[0];
    L_Last_Written_Persist_Buffer[1] := L_Persist_Buffer[1];
    L_Last_Written_Persist_Buffer[2] := L_Persist_Buffer[2];
    L_Last_Written_Persist_Buffer[3] := L_Persist_Buffer[3];
    L_Last_Written_Persist_Buffer[4] := L_Persist_Buffer[4];
    L_Last_Persist_Write_MS := GVL_STATUS.G_System_Time_MS;
END_IF;

// 15. Черный ящик
L_BB_Record.Timestamp := GVL_STATUS.G_System_Time_MS;
L_BB_Record.PLC_Active_ID := GVL_STATUS.G_PLC_ID;
L_BB_Record.Gas_Methane_LEL := GVL_STATE.G_Methane_Sensors[1];
L_BB_Record.Gas_CO_PPM := GVL_STATE.G_CO_Sensors[1];
L_BB_Record.Flood_Active := GVL_ALARM.G_Flood_Alarm_Active;
L_BB_Record.Fire_Active := GVL_ALARM.G_Fire_Alarm_Active;
L_BB_Record.Valve_Gas_Status := SEL(GVL_COMMAND.G_Gas_Valve_Close, BYTE#0, BYTE#1);
L_BB_Record.Valve_Water_Status := SEL((GVL_COMMAND.G_Close_Valve_35 OR GVL_COMMAND.G_Close_Valve_36), BYTE#0, BYTE#1);

L_BB_Record.System_Mode := TO_BYTE(TO_INT(GVL_STATE.G_System_Mode));
L_BB_Record.First_Fault_Type := TO_BYTE(TO_INT(fbSystemHealth.VO_First_Fault_Type));
L_BB_Record.First_Fault_Source := TO_BYTE(TO_INT(fbSystemHealth.VO_First_Fault_Source));
L_BB_Record.First_Fault_Active := fbSystemHealth.VO_First_Fault_Active;
L_BB_Record.System_Severity := TO_BYTE(TO_INT(fbSystemHealth.VO_System_Severity));
L_BB_Record.Root_Cause := TO_BYTE(TO_INT(fbSystemHealth.VO_Root_Cause));
L_BB_Record.Watchdog_Fault := fbWatchdog.VO_Watchdog_Fault;

L_BB_Freeze := GVL_ALARM.G_Gas_Alarm_Active OR GVL_ALARM.G_Fire_Alarm_Active OR GVL_ALARM.G_Flood_Alarm_Active OR fbSystemHealth.VO_First_Fault_Active;

fbBlackBox(
    VI_Current_Data := L_BB_Record,
    VI_Freeze := L_BB_Freeze
);

// 15.1. Менеджер истории / diagnostics bridge
L_History_Write_Event := FALSE;
L_History_Event.timestamp_ms := GVL_STATUS.G_System_Time_MS;
L_History_Event.event_code := 0;
L_History_Event.event_value := 0.0;
L_History_Event.unit := 0;
L_History_Event.zone_id := 0;
L_History_Event.operator_id := 'SYSTEM';
L_History_Event.priority := E_ALERT_PRIORITY.ALERT_PRIORITY_HIGH;

IF GVL_STATE.G_System_Mode <> L_Last_System_Mode THEN
    L_History_Write_Event := TRUE;
    L_History_Event.event_code := 1101; // System mode transition
    L_History_Event.event_value := TO_REAL(TO_INT(GVL_STATE.G_System_Mode));
    L_History_Event.unit := 1; // system mode domain
    L_History_Event.zone_id := 0;
    IF GVL_STATE.G_System_Mode = E_System_Operating_Mode.MODE_NORMAL THEN
        L_History_Event.priority := E_ALERT_PRIORITY.ALERT_PRIORITY_HIGH;
    ELSE
        L_History_Event.priority := E_ALERT_PRIORITY.ALERT_PRIORITY_HIGH;
    END_IF;
    L_Last_System_Mode := GVL_STATE.G_System_Mode;

ELSIF fbSystemHealth.VO_Root_Cause <> L_Last_Root_Cause THEN
    L_History_Write_Event := TRUE;
    L_History_Event.event_code := 1102; // Root cause changed
    L_History_Event.event_value := TO_REAL(TO_INT(fbSystemHealth.VO_Root_Cause));
    L_History_Event.unit := 2; // root cause enum domain
    L_History_Event.zone_id := TO_BYTE(fbSystemHealth.VO_First_Fault_Source);
    L_History_Event.priority := E_ALERT_PRIORITY.ALERT_PRIORITY_HIGH;
    L_Last_Root_Cause := fbSystemHealth.VO_Root_Cause;

ELSIF fbSystemHealth.VO_First_Fault_Source <> L_Last_First_Fault_Source THEN
    L_History_Write_Event := TRUE;
    L_History_Event.event_code := 1103; // First fault source changed
    L_History_Event.event_value := TO_REAL(fbSystemHealth.VO_First_Fault_Source);
    L_History_Event.unit := 3; // root cause source domain
    L_History_Event.zone_id := TO_BYTE(fbSystemHealth.VO_First_Fault_Source);
    L_History_Event.priority := E_ALERT_PRIORITY.ALERT_PRIORITY_HIGH;
    L_Last_First_Fault_Source := fbSystemHealth.VO_First_Fault_Source;

ELSIF GVL_STATUS.G_Current_Scenario <> GVL_STATUS.G_Previous_Scenario THEN
    L_History_Write_Event := TRUE;
    L_History_Event.event_code := 1001; // Scenario transition
    L_History_Event.event_value := TO_REAL(GVL_STATUS.G_Current_Scenario);
    L_History_Event.unit := 4; // scenario domain
    L_History_Event.zone_id := 0;
    L_History_Event.priority := E_ALERT_PRIORITY.ALERT_PRIORITY_HIGH;

    fbLogEvent(
        VI_Event_Type := 1,
        VI_Timestamp := GVL_STATUS.G_System_Time_MS,
        VI_Param1 := TO_UDINT(L_Scenario_Source),
        VI_Param2 := TO_UDINT(GVL_STATUS.G_Current_Scenario)
    );

    GVL_STATUS.G_Previous_Scenario := GVL_STATUS.G_Current_Scenario;

ELSIF GVL_STATUS.G_Diagnostics.Alarm_Event_Pulse THEN
    L_History_Write_Event := TRUE;
    L_History_Event.event_code := TO_WORD(GVL_STATUS.G_Diagnostics.Alarm_Event_Code);
    L_History_Event.event_value := GVL_STATUS.G_Diagnostics.Alarm_Event_Value;
    L_History_Event.unit := 10; // alarm lifecycle domain
    L_History_Event.zone_id := 0;
    L_History_Event.priority := E_ALERT_PRIORITY.ALERT_PRIORITY_HIGH;

ELSIF GVL_STATUS.G_Diagnostics.Operator_Journal_Event_Seq <> L_Last_Operator_Journal_Seq THEN
    L_History_Write_Event := TRUE;
    L_History_Event.event_code := 1301; // Operator journal event
    L_History_Event.event_value := TO_REAL(GVL_STATUS.G_Diagnostics.Operator_Journal_Event_Seq);
    L_History_Event.unit := 20; // operator journal domain
    L_History_Event.zone_id := 0;
    L_History_Event.priority := E_ALERT_PRIORITY.ALERT_PRIORITY_HIGH;
    L_Last_Operator_Journal_Seq := GVL_STATUS.G_Diagnostics.Operator_Journal_Event_Seq;
END_IF;

// --- History anti-flood / dedup ---
IF L_History_Write_Event THEN
    IF (L_History_Event.event_code = L_Last_Event_Code)
       AND (ABS(L_History_Event.event_value - L_Last_Event_Value) < 0.001)
       AND (GVL_STATUS.G_System_Time_MS - L_Last_Event_Time_MS < 5000) THEN
        L_History_Write_Event := FALSE;
    ELSE
        L_Last_Event_Code := L_History_Event.event_code;
        L_Last_Event_Value := L_History_Event.event_value;
        L_Last_Event_Time_MS := GVL_STATUS.G_System_Time_MS;
    END_IF;
END_IF;

fbHistoryManager(
    VI_System_Time_MS := GVL_STATUS.G_System_Time_MS,
    VI_Write_Event := L_History_Write_Event,
    VI_Event := L_History_Event
);

L_Maintenance_Apply_Intent := FALSE;

// Dangerous action confirmation flow
IF GVL_COMMAND.CMD_Dangerous_Action_Request AND
   NOT L_Dangerous_Action_Request_Prev AND
   (GVL_COMMAND.CMD_User_Access_Level >= 2) THEN

    IF NOT L_Dangerous_Action_Armed THEN
        fbLogEvent(
            VI_Event_Type := 8,
            VI_Timestamp := GVL_STATUS.G_System_Time_MS,
            VI_Param1 := TO_UDINT(GVL_COMMAND.CMD_User_Access_Level),
            VI_Param2 := 1
        );
    END_IF;

    L_Dangerous_Action_Armed := TRUE;
    L_Dangerous_Action_Deadline_MS := GVL_STATUS.G_System_Time_MS + 15000;
    GVL_STATUS.G_Diagnostics.Dangerous_Action_Pending_Confirm := TRUE;
    GVL_STATUS.G_Diagnostics.Dangerous_Action_Confirm_Deadline_MS := L_Dangerous_Action_Deadline_MS;
    GVL_STATUS.G_Diagnostics.Dangerous_Action_Confirm_Text := 'Подтвердите опасное действие в течение 15 секунд';
END_IF;
IF L_Dangerous_Action_Armed AND (GVL_STATUS.G_System_Time_MS > L_Dangerous_Action_Deadline_MS) THEN
    L_Dangerous_Action_Armed := FALSE;
    L_Maintenance_Apply_Intent := FALSE;
    GVL_STATUS.G_Diagnostics.Dangerous_Action_Pending_Confirm := FALSE;
    GVL_STATUS.G_Diagnostics.Dangerous_Action_Confirm_Text := 'Окно подтверждения истекло';
END_IF;
IF GVL_COMMAND.CMD_Dangerous_Action_Confirm AND
   L_Dangerous_Action_Armed AND
   (GVL_COMMAND.CMD_User_Access_Level >= 2) THEN
    L_Maintenance_Apply_Intent := TRUE;

    fbLogEvent(
        VI_Event_Type := 9,
        VI_Timestamp := GVL_STATUS.G_System_Time_MS,
        VI_Param1 := TO_UDINT(GVL_COMMAND.CMD_User_Access_Level),
        VI_Param2 := 1
    );

    L_Dangerous_Action_Armed := FALSE;
    GVL_STATUS.G_Diagnostics.Dangerous_Action_Pending_Confirm := FALSE;
    GVL_STATUS.G_Diagnostics.Dangerous_Action_Confirm_Text := 'Опасное действие подтверждено оператором';
END_IF;

// HMI maintenance mode control (confirmation-aware)
IF L_Maintenance_Apply_Intent AND
   ((GVL_STATE.G_System_Mode = E_System_Operating_Mode.MODE_NORMAL) OR
    (GVL_STATE.G_System_Mode = E_System_Operating_Mode.MODE_DEGRADED)) THEN
    FOR L_i := 1 TO GVL_CONSTANTS.C_MAX_MANIFOLDS DO
        GVL_CONFIG.G_Manifold_Pump_In_Service[L_i] := GVL_COMMAND.CMD_Set_Manifold_Pump_In_Service[L_i];
    END_FOR;
    GVL_CONFIG.G_DHW_Heating_Pump_In_Service := GVL_COMMAND.CMD_Set_DHW_Heating_Pump_In_Service;
    GVL_CONFIG.G_DHW_Circ_Pump_In_Service := GVL_COMMAND.CMD_Set_DHW_Circ_Pump_In_Service;
END_IF;

// Access level enforcement for dangerous actions
GVL_STATUS.G_Diagnostics.User_Access_Level_Active := GVL_COMMAND.CMD_User_Access_Level;
GVL_STATUS.G_Diagnostics.User_Access_Denied := FALSE;
GVL_STATUS.G_Diagnostics.User_Access_Deny_Reason := '';
GVL_STATUS.G_Diagnostics.Operator_Action_Blocked := FALSE;
GVL_STATUS.G_Diagnostics.Operator_Block_Reason := '';
IF GVL_COMMAND.CMD_Dangerous_Action_Request OR GVL_COMMAND.CMD_Dangerous_Action_Confirm THEN
    IF GVL_COMMAND.CMD_User_Access_Level < 2 THEN
        IF NOT L_User_Access_Denied_Prev THEN
            fbLogEvent(
                VI_Event_Type := 10,
                VI_Timestamp := GVL_STATUS.G_System_Time_MS,
                VI_Param1 := TO_UDINT(GVL_COMMAND.CMD_User_Access_Level),
                VI_Param2 := 2
            );
        END_IF;

        GVL_STATUS.G_Diagnostics.User_Access_Denied := TRUE;
        GVL_STATUS.G_Diagnostics.User_Access_Deny_Reason := 'Недостаточный уровень доступа для опасного действия';
        GVL_STATUS.G_Diagnostics.Operator_Action_Blocked := TRUE;
        GVL_STATUS.G_Diagnostics.Operator_Block_Reason := 'Требуется уровень ENGINEER для опасного действия';
        L_Dangerous_Action_Armed := FALSE;
        GVL_STATUS.G_Diagnostics.Dangerous_Action_Pending_Confirm := FALSE;
        GVL_STATUS.G_Diagnostics.Dangerous_Action_Confirm_Text := 'Доступ запрещён: требуется уровень ENGINEER';
    END_IF;
END_IF;

L_User_Access_Denied_Prev := GVL_STATUS.G_Diagnostics.User_Access_Denied;
L_Dangerous_Action_Request_Prev := GVL_COMMAND.CMD_Dangerous_Action_Request;

// Hard revert for forbidden operator actions
IF GVL_STATUS.G_Diagnostics.Operator_Action_Blocked THEN
    FOR L_i := 1 TO GVL_CONSTANTS.C_MAX_MANIFOLDS DO
        IF NOT GVL_CONFIG.G_Manifold_Pump_In_Service[L_i] THEN
            GVL_CONFIG.G_Manifold_Pump_In_Service[L_i] := TRUE;
        END_IF;
    END_FOR;
    IF NOT GVL_CONFIG.G_DHW_Heating_Pump_In_Service THEN
        GVL_CONFIG.G_DHW_Heating_Pump_In_Service := TRUE;
    END_IF;
    IF NOT GVL_CONFIG.G_DHW_Circ_Pump_In_Service THEN
        GVL_CONFIG.G_DHW_Circ_Pump_In_Service := TRUE;
    END_IF;
    GVL_STATUS.G_Diagnostics.Operator_Last_Forbidden_Action := GVL_STATUS.G_Diagnostics.Operator_Block_Reason;
END_IF;

// Operator action journal
IF GVL_STATUS.G_Diagnostics.Operator_Action_Blocked AND NOT L_Last_Operator_Blocked THEN
    GVL_STATUS.G_Diagnostics.Operator_Journal_Event_Seq := GVL_STATUS.G_Diagnostics.Operator_Journal_Event_Seq + 1;
END_IF;
L_Last_Operator_Blocked := GVL_STATUS.G_Diagnostics.Operator_Action_Blocked;
IF GVL_CONFIG.G_DHW_Heating_Pump_In_Service <> L_Last_DHW_Heating_In_Service THEN
    IF GVL_CONFIG.G_DHW_Heating_Pump_In_Service THEN
        GVL_STATUS.G_Diagnostics.Maintenance_Last_Action := 'Насос загрузки ГВС возвращён из ТО';
        IF L_Last_Maintenance_Action_Code <> 1101 THEN
            GVL_STATUS.G_Diagnostics.Operator_Journal_Event_Seq := GVL_STATUS.G_Diagnostics.Operator_Journal_Event_Seq + 1;
            L_Last_Maintenance_Action_Code := 1101;
        END_IF;
    ELSE
        GVL_STATUS.G_Diagnostics.Maintenance_Last_Action := 'Насос загрузки ГВС выведен в ТО';
        IF L_Last_Maintenance_Action_Code <> 1102 THEN
            GVL_STATUS.G_Diagnostics.Operator_Journal_Event_Seq := GVL_STATUS.G_Diagnostics.Operator_Journal_Event_Seq + 1;
            L_Last_Maintenance_Action_Code := 1102;
        END_IF;
    END_IF;
END_IF;
L_Last_DHW_Heating_In_Service := GVL_CONFIG.G_DHW_Heating_Pump_In_Service;
IF GVL_CONFIG.G_DHW_Circ_Pump_In_Service <> L_Last_DHW_Circ_In_Service THEN
    IF GVL_CONFIG.G_DHW_Circ_Pump_In_Service THEN
        GVL_STATUS.G_Diagnostics.Maintenance_Last_Action := 'Насос рециркуляции ГВС возвращён из ТО';
        IF L_Last_Maintenance_Action_Code <> 1201 THEN
            GVL_STATUS.G_Diagnostics.Operator_Journal_Event_Seq := GVL_STATUS.G_Diagnostics.Operator_Journal_Event_Seq + 1;
            L_Last_Maintenance_Action_Code := 1201;
        END_IF;
    ELSE
        GVL_STATUS.G_Diagnostics.Maintenance_Last_Action := 'Насос рециркуляции ГВС выведен в ТО';
        IF L_Last_Maintenance_Action_Code <> 1202 THEN
            GVL_STATUS.G_Diagnostics.Operator_Journal_Event_Seq := GVL_STATUS.G_Diagnostics.Operator_Journal_Event_Seq + 1;
            L_Last_Maintenance_Action_Code := 1202;
        END_IF;
    END_IF;
END_IF;
L_Last_DHW_Circ_In_Service := GVL_CONFIG.G_DHW_Circ_Pump_In_Service;
IF GVL_STATUS.G_Diagnostics.Operator_Journal_Event_Seq <> GVL_STATUS.G_Diagnostics.Operator_Journal_Last_Seq THEN
    GVL_STATUS.G_Diagnostics.Operator_Journal_3 := GVL_STATUS.G_Diagnostics.Operator_Journal_2;
    GVL_STATUS.G_Diagnostics.Operator_Journal_2 := GVL_STATUS.G_Diagnostics.Operator_Journal_1;
    IF GVL_STATUS.G_Diagnostics.Operator_Last_Forbidden_Action <> '' THEN
        GVL_STATUS.G_Diagnostics.Operator_Journal_1 := GVL_STATUS.G_Diagnostics.Operator_Last_Forbidden_Action;
    ELSE
        GVL_STATUS.G_Diagnostics.Operator_Journal_1 := GVL_STATUS.G_Diagnostics.Maintenance_Last_Action;
    END_IF;
    GVL_STATUS.G_Diagnostics.Operator_Journal_Last_Seq := GVL_STATUS.G_Diagnostics.Operator_Journal_Event_Seq;
END_IF;

// ========================================
// CoreKernel live observer (diagnostic only)
// ========================================
// fbCoreKernelObserver disabled temporarily

// === NVRAM SNAPSHOT VIA STRUCT ADAPTER ===
L_Persist_Struct.System_Mode := GVL_STATE.G_System_Mode;

L_Persist_Struct.Safety_Gas_Latched := GVL_STATE.G_Safety_Gas_Latched;
L_Persist_Struct.Safety_Smoke_Latched := GVL_STATE.G_Safety_Smoke_Latched;
L_Persist_Struct.Safety_Leak_Latched := GVL_STATE.G_Safety_Leak_Latched;

L_Persist_Struct.DHW_Heating_Pump := GVL_STATE.G_DHW_Heating_Pump;
L_Persist_Struct.Valid := TRUE;

// mirror to legacy persistent variables
GVL_PERSISTENT.P_System_Mode := L_Persist_Struct.System_Mode;

GVL_PERSISTENT.P_Safety_Gas_Latched := L_Persist_Struct.Safety_Gas_Latched;
GVL_PERSISTENT.P_Safety_Smoke_Latched := L_Persist_Struct.Safety_Smoke_Latched;
GVL_PERSISTENT.P_Safety_Leak_Latched := L_Persist_Struct.Safety_Leak_Latched;

GVL_PERSISTENT.P_DHW_Heating_Active := L_Persist_Struct.DHW_Heating_Pump;
GVL_PERSISTENT.P_Valid := L_Persist_Struct.Valid;

// === TREND EXECUTION (SAFE MVP) ===
L_Trend_Data.config.param_type := 1;
L_Trend_Data.config.zone_id := 0;
L_Trend_Data.config.enabled := TRUE;
L_Trend_Data.config.deviation_threshold_percent := 1.0;
L_Trend_Data.config.history_days := 1;

L_Trend_Logger(
    VI_System_Time_MS := GVL_STATUS.G_System_Time_MS,
    VI_Config := L_Trend_Data.config,
    VI_Current_Value := GVL_STATE.G_Outdoor_Temp
);

L_Trend_Data := L_Trend_Logger.VO_Data;

// === TREND ANALYSIS VIA ADAPTER ===
L_Trend_Adapter(
    VI_Data := L_Trend_Data,
    VO_Average => L_Trend_Avg,
    VO_Min => L_Trend_Min,
    VO_Max => L_Trend_Max,
    VO_Trend_Up => L_Trend_Up,
    VO_Trend_Down => L_Trend_Down
);

// === TREND MULTI-SIGNAL FOUNDATION ===
// Channel 1 is currently active (Outdoor Temp / TEMP_AIR).
// Channel 2 reserved for future integration.
// HMI may use GVL_Trend.G_Trend_Selected_Channel to switch active graph source.

// === TREND → GVL FOR HMI ===

// === TREND BUFFER UPDATE ===

// === TREND CHANNEL 2 (FLOOR TEMP, SHARED INDEX) ===
IF GVL_Trend.G_Trend_Channel2_Enabled THEN

    GVL_Trend.G_Trend_Buffer_2_Index := GVL_Trend.G_Trend_Buffer_Index;
    GVL_Trend.G_Trend_Buffer_2[GVL_Trend.G_Trend_Buffer_2_Index] := L_FloorTemps_8[1];
    GVL_Trend.G_Trend_Buffer_2_Timestamps[GVL_Trend.G_Trend_Buffer_2_Index] := GVL_STATUS.G_System_Time_MS;

    IF GVL_Trend.G_Trend_Buffer_2_Valid_Count < 50 THEN
        GVL_Trend.G_Trend_Buffer_2_Valid_Count := GVL_Trend.G_Trend_Buffer_2_Valid_Count + 1;
    ELSE
        GVL_Trend.G_Trend_Buffer_2_Is_Wrapped := TRUE;
    END_IF;

    GVL_Trend.G_Trend_Channel2_Param_Type := 2; // TEMP_FLOOR

END_IF;

// === TREND META UPDATE ===
GVL_Trend.G_Trend_Last_Update_MS := GVL_STATUS.G_System_Time_MS;
GVL_Trend.G_Trend_Param_Type := 1; // TEMP_AIR (пока фикс)

IF GVL_Trend.G_Trend_Valid_Count < 50 THEN
    GVL_Trend.G_Trend_Valid_Count := GVL_Trend.G_Trend_Valid_Count + 1;
ELSE
    GVL_Trend.G_Trend_Is_Wrapped := TRUE;
END_IF;

GVL_Trend.G_Trend_Buffer_Index := GVL_Trend.G_Trend_Buffer_Index + 1;
IF GVL_Trend.G_Trend_Buffer_Index > 50 THEN
    GVL_Trend.G_Trend_Buffer_Index := 1;
END_IF;

GVL_Trend.G_Trend_Buffer[GVL_Trend.G_Trend_Buffer_Index] := L_Trend_Avg;
GVL_Trend.G_Trend_Buffer_Timestamps[GVL_Trend.G_Trend_Buffer_Index] := GVL_STATUS.G_System_Time_MS;

GVL_Trend.G_Trend_Avg := L_Trend_Avg;
GVL_Trend.G_Trend_Min := L_Trend_Min;
GVL_Trend.G_Trend_Max := L_Trend_Max;
GVL_Trend.G_Trend_Up := L_Trend_Up;
GVL_Trend.G_Trend_Down := L_Trend_Down;

// === TREND HMI NORMALIZATION ===
IF GVL_Trend.G_Trend_Selected_Channel = 2 AND GVL_Trend.G_Trend_Channel2_Enabled THEN
    GVL_Trend.G_Trend_Active_Param_Type := GVL_Trend.G_Trend_Channel2_Param_Type;
    GVL_Trend.G_Trend_Active_Label := GVL_Trend.G_Trend_Channel2_Label;
ELSE
    GVL_Trend.G_Trend_Active_Param_Type := GVL_Trend.G_Trend_Param_Type;
    GVL_Trend.G_Trend_Active_Label := GVL_Trend.G_Trend_Channel1_Label;
END_IF;

// === TREND ACTIVE VIEW FOR HMI ===
IF GVL_Trend.G_Trend_Selected_Channel = 2 AND GVL_Trend.G_Trend_Channel2_Enabled THEN
    GVL_Trend.G_Trend_Active_Index := GVL_Trend.G_Trend_Buffer_2_Index;
    GVL_Trend.G_Trend_Active_Valid_Count := GVL_Trend.G_Trend_Buffer_2_Valid_Count;
    GVL_Trend.G_Trend_Active_Is_Wrapped := GVL_Trend.G_Trend_Buffer_2_Is_Wrapped;

    IF GVL_Trend.G_Trend_Buffer_2_Index >= 1 AND GVL_Trend.G_Trend_Buffer_2_Index <= 50 THEN
        GVL_Trend.G_Trend_Active_Value := GVL_Trend.G_Trend_Buffer_2[GVL_Trend.G_Trend_Buffer_2_Index];
        GVL_Trend.G_Trend_Active_Timestamp := GVL_Trend.G_Trend_Buffer_2_Timestamps[GVL_Trend.G_Trend_Buffer_2_Index];
    END_IF;
ELSE
    GVL_Trend.G_Trend_Active_Index := GVL_Trend.G_Trend_Buffer_Index;
    GVL_Trend.G_Trend_Active_Valid_Count := GVL_Trend.G_Trend_Valid_Count;
    GVL_Trend.G_Trend_Active_Is_Wrapped := GVL_Trend.G_Trend_Is_Wrapped;

    IF GVL_Trend.G_Trend_Buffer_Index >= 1 AND GVL_Trend.G_Trend_Buffer_Index <= 50 THEN
        GVL_Trend.G_Trend_Active_Value := GVL_Trend.G_Trend_Buffer[GVL_Trend.G_Trend_Buffer_Index];
        GVL_Trend.G_Trend_Active_Timestamp := GVL_Trend.G_Trend_Buffer_Timestamps[GVL_Trend.G_Trend_Buffer_Index];
    END_IF;
END_IF;

// === SENSOR PROCESSING (SHADOW EXEC) ===
fbSensorCO(
    VI_Raw_Value := REAL_TO_WORD(GVL_STATE.G_CO_Sensors[1]),
    VI_Sensor_Type := 0,
    VI_Min_Scale := 0.0,
    VI_Max_Scale := 100.0,
    VI_Offset := 0.0,
    VI_System_Time_MS := GVL_STATUS.G_System_Time_MS
);
L_CO_Processed := fbSensorCO.VO_Value;

fbCalibCO(
    VI_Raw_Value := L_CO_Processed,
    VI_Record := GVL_CONFIG.G_HMI_Sensor_Calibrations[1]
);
L_CO_Calibrated := fbCalibCO.VO_Calibrated_Value;

// === SHADOW EXPORT ===
GVL_Sensor_Shadow.G_CO_Raw := GVL_STATE.G_CO_Sensors[1];
GVL_Sensor_Shadow.G_CO_Processed := L_CO_Processed;
GVL_Sensor_Shadow.G_CO_Calibrated := L_CO_Calibrated;
GVL_Sensor_Shadow.G_CO_Error := fbSensorCO.VO_Error;
GVL_Sensor_Shadow.G_CO_Diag_Code := fbSensorCO.VO_Diag_Code;

// === METHANE SHADOW EXEC ===
fbSensorMethane(
    VI_Raw_Value := REAL_TO_WORD(GVL_STATE.G_Methane_Sensors[1]),
    VI_Sensor_Type := 0,
    VI_Min_Scale := 0.0,
    VI_Max_Scale := 100.0,
    VI_Offset := 0.0,
    VI_System_Time_MS := GVL_STATUS.G_System_Time_MS
);
L_Methane_Processed := fbSensorMethane.VO_Value;

fbCalibMethane(
    VI_Raw_Value := L_Methane_Processed,
    VI_Record := GVL_CONFIG.G_HMI_Sensor_Calibrations[2]
);
L_Methane_Calibrated := fbCalibMethane.VO_Calibrated_Value;

// === METHANE SHADOW EXPORT ===
GVL_Sensor_Shadow.G_Methane_Raw := GVL_STATE.G_Methane_Sensors[1];
GVL_Sensor_Shadow.G_Methane_Processed := L_Methane_Processed;
GVL_Sensor_Shadow.G_Methane_Calibrated := L_Methane_Calibrated;
GVL_Sensor_Shadow.G_Methane_Error := fbSensorMethane.VO_Error;
GVL_Sensor_Shadow.G_Methane_Diag_Code := fbSensorMethane.VO_Diag_Code;

// === SMOKE SHADOW EXEC ===
fbSmokeDetector(
    VI_Smoke_Signal := GVL_STATE.G_Smoke_Sensors[1]
);
L_Smoke_Detected := fbSmokeDetector.VO_Smoke_Detected;

// === SMOKE SHADOW EXPORT ===
GVL_Sensor_Shadow.G_Smoke_Raw := GVL_STATE.G_Smoke_Sensors[1];
GVL_Sensor_Shadow.G_Smoke_Detected := L_Smoke_Detected;

// === SAFETY SHADOW VS RUNTIME BRIDGE ===

// CO
GVL_Safety_Bridge.G_CO_Runtime := GVL_STATE.G_CO_Sensors[1];
GVL_Safety_Bridge.G_CO_Shadow  := GVL_Sensor_Shadow.G_CO_Calibrated;
GVL_Safety_Bridge.G_CO_Diff    := ABS(GVL_Safety_Bridge.G_CO_Runtime - GVL_Safety_Bridge.G_CO_Shadow);

// METHANE
GVL_Safety_Bridge.G_Methane_Runtime := GVL_STATE.G_Methane_Sensors[1];
GVL_Safety_Bridge.G_Methane_Shadow  := GVL_Sensor_Shadow.G_Methane_Calibrated;
GVL_Safety_Bridge.G_Methane_Diff    := ABS(GVL_Safety_Bridge.G_Methane_Runtime - GVL_Safety_Bridge.G_Methane_Shadow);

// SMOKE
GVL_Safety_Bridge.G_Smoke_Runtime := GVL_STATE.G_Smoke_Sensors[1];
GVL_Safety_Bridge.G_Smoke_Shadow  := GVL_Sensor_Shadow.G_Smoke_Detected;
GVL_Safety_Bridge.G_Smoke_Diff    := GVL_Safety_Bridge.G_Smoke_Runtime XOR GVL_Safety_Bridge.G_Smoke_Shadow;

// === SAFETY SELECTOR LAYER ===
GVL_Safety_Selector.G_Use_Shadow_Methane := TRUE;
GVL_Safety_Selector.G_Use_Shadow_Smoke := TRUE;
GVL_Safety_Selector.G_Use_Shadow_CO := TRUE;

// base copy from runtime arrays
FOR L_Safety_Selector_i := 1 TO GVL_CONSTANTS.C_MAX_CO_SENSORS DO
    GVL_Safety_Selector.G_CO_Effective_Array[L_Safety_Selector_i] := GVL_STATE.G_CO_Sensors[L_Safety_Selector_i];
END_FOR;

FOR L_Safety_Selector_i := 1 TO GVL_CONSTANTS.C_MAX_METHANE_SENSORS DO
    GVL_Safety_Selector.G_Methane_Effective_Array[L_Safety_Selector_i] := GVL_STATE.G_Methane_Sensors[L_Safety_Selector_i];
END_FOR;

FOR L_Safety_Selector_i := 1 TO GVL_CONSTANTS.C_MAX_SMOKE_SENSORS DO
    GVL_Safety_Selector.G_Smoke_Effective_Array[L_Safety_Selector_i] := GVL_STATE.G_Smoke_Sensors[L_Safety_Selector_i];
END_FOR;

// CO
IF GVL_Safety_Selector.G_Use_Shadow_CO THEN
    GVL_Safety_Selector.G_CO_Effective := GVL_Sensor_Shadow.G_CO_Calibrated;
    GVL_Safety_Selector.G_CO_Effective_Array[1] := GVL_Sensor_Shadow.G_CO_Calibrated;
ELSE
    GVL_Safety_Selector.G_CO_Effective := GVL_STATE.G_CO_Sensors[1];
END_IF;

// METHANE
IF GVL_Safety_Selector.G_Use_Shadow_Methane THEN
    GVL_Safety_Selector.G_Methane_Effective := GVL_Sensor_Shadow.G_Methane_Calibrated;
    GVL_Safety_Selector.G_Methane_Effective_Array[1] := GVL_Sensor_Shadow.G_Methane_Calibrated;
ELSE
    GVL_Safety_Selector.G_Methane_Effective := GVL_STATE.G_Methane_Sensors[1];
END_IF;

// SMOKE
IF GVL_Safety_Selector.G_Use_Shadow_Smoke THEN
    GVL_Safety_Selector.G_Smoke_Effective := GVL_Sensor_Shadow.G_Smoke_Detected;
    GVL_Safety_Selector.G_Smoke_Effective_Array[1] := GVL_Sensor_Shadow.G_Smoke_Detected;
ELSE
    GVL_Safety_Selector.G_Smoke_Effective := GVL_STATE.G_Smoke_Sensors[1];
END_IF;

// === SHADOW METHANE/SMOKE DIAGNOSTIC EXPORT ===
GVL_STATUS.G_Diagnostics.Sensor_Shadow_Methane_Active := GVL_Safety_Selector.G_Use_Shadow_Methane;
GVL_STATUS.G_Diagnostics.Sensor_Shadow_Methane_Diff := GVL_Safety_Bridge.G_Methane_Diff;
GVL_STATUS.G_Diagnostics.Sensor_Shadow_Smoke_Active := GVL_Safety_Selector.G_Use_Shadow_Smoke;

IF GVL_Safety_Selector.G_Use_Shadow_Methane THEN
    GVL_STATUS.G_Diagnostics.Sensor_Shadow_Methane_Status_Text := 'Methane shadow ACTIVE';
ELSE
    GVL_STATUS.G_Diagnostics.Sensor_Shadow_Methane_Status_Text := 'Methane shadow OFF';
END_IF;

IF GVL_Safety_Selector.G_Use_Shadow_Smoke THEN
    GVL_STATUS.G_Diagnostics.Sensor_Shadow_Smoke_Status_Text := 'Smoke shadow ACTIVE';
ELSE
    GVL_STATUS.G_Diagnostics.Sensor_Shadow_Smoke_Status_Text := 'Smoke shadow OFF';
END_IF;

// === SHADOW CO DIAGNOSTIC EXPORT ===
GVL_STATUS.G_Diagnostics.Sensor_Shadow_CO_Active := GVL_Safety_Selector.G_Use_Shadow_CO;
GVL_STATUS.G_Diagnostics.Sensor_Shadow_CO_Diff := GVL_Safety_Bridge.G_CO_Diff;

IF GVL_Safety_Selector.G_Use_Shadow_CO THEN
    GVL_STATUS.G_Diagnostics.Sensor_Shadow_CO_Status_Text := 'CO shadow ACTIVE';
ELSE
    GVL_STATUS.G_Diagnostics.Sensor_Shadow_CO_Status_Text := 'CO shadow OFF';
END_IF;

// === SHADOW SAFETY QUALITY FLAGS ===
GVL_STATUS.G_Diagnostics.Sensor_Shadow_CO_Unstable :=
    GVL_Safety_Bridge.G_CO_Diff > GVL_Safety_Selector.G_CO_Shadow_Max_Diff;

GVL_STATUS.G_Diagnostics.Sensor_Shadow_Methane_Unstable :=
    GVL_Safety_Bridge.G_Methane_Diff > GVL_Safety_Selector.G_Methane_Shadow_Max_Diff;

GVL_STATUS.G_Diagnostics.Sensor_Shadow_Smoke_Mismatch :=
    GVL_Safety_Bridge.G_Smoke_Diff;

// === SHADOW SAFETY POLICY ===
IF GVL_Safety_Selector.G_Block_Shadow_On_Mismatch THEN
    IF GVL_STATUS.G_Diagnostics.Sensor_Shadow_CO_Unstable THEN
        GVL_Safety_Selector.G_Use_Shadow_CO := FALSE;
    END_IF;

    IF GVL_STATUS.G_Diagnostics.Sensor_Shadow_Methane_Unstable THEN
        GVL_Safety_Selector.G_Use_Shadow_Methane := FALSE;
    END_IF;

    IF GVL_STATUS.G_Diagnostics.Sensor_Shadow_Smoke_Mismatch THEN
        GVL_Safety_Selector.G_Use_Shadow_Smoke := FALSE;
    END_IF;
END_IF;

IF GVL_STATUS.G_Diagnostics.Sensor_Shadow_Smoke_Mismatch THEN
    GVL_STATUS.G_Diagnostics.Sensor_Shadow_Quality_Text := 'Smoke shadow mismatch';
ELSIF GVL_STATUS.G_Diagnostics.Sensor_Shadow_Methane_Unstable THEN
    GVL_STATUS.G_Diagnostics.Sensor_Shadow_Quality_Text := 'Methane shadow unstable';
ELSIF GVL_STATUS.G_Diagnostics.Sensor_Shadow_CO_Unstable THEN
    GVL_STATUS.G_Diagnostics.Sensor_Shadow_Quality_Text := 'CO shadow unstable';
ELSE
    GVL_STATUS.G_Diagnostics.Sensor_Shadow_Quality_Text := 'Shadow safety quality OK';
END_IF;

// === LIFETIME UPDATE ===

// pump (временно FALSE — до реального сигнала)
fbLifetimePump(
    VI_System_Time_MS := GVL_STATUS.G_System_Time_MS,
    VI_Device_Active  := GVL_PERSISTENT.P_DHW_Heating_Active,
    VI_Device_ID      := GVL_Lifetime.G_Device_Pump,
    VI_Nominal_Hours  := GVL_Lifetime.G_Pump_Nominal_Hours,
    VIO_Status        := GVL_Lifetime.G_Status[1]
);

// fan (временно FALSE — до реального сигнала)
fbLifetimeFan(
    VI_System_Time_MS := GVL_STATUS.G_System_Time_MS,
    VI_Device_Active  := (
        GVL_STATE.G_Supply_Fans[1] > 0 OR
        GVL_STATE.G_Exhaust_Fans[1] > 0
    ),
    VI_Device_ID      := GVL_Lifetime.G_Device_Fan,
    VI_Nominal_Hours  := GVL_Lifetime.G_Fan_Nominal_Hours,
    VIO_Status        := GVL_Lifetime.G_Status[2]
);

// === LIFETIME HMI ACTIVE VIEW ===
IF GVL_Lifetime.G_Active_Device_Index < 1 THEN
    GVL_Lifetime.G_Active_Device_Index := 1;
ELSIF GVL_Lifetime.G_Active_Device_Index > 4 THEN
    GVL_Lifetime.G_Active_Device_Index := 4;
END_IF;

GVL_Lifetime.G_Active_Runtime_Hours := GVL_Lifetime.G_Status[GVL_Lifetime.G_Active_Device_Index].runtime_hours;
GVL_Lifetime.G_Active_Remaining_Hours := GVL_Lifetime.G_Status[GVL_Lifetime.G_Active_Device_Index].remaining_hours;
GVL_Lifetime.G_Active_Remaining_Percent := GVL_Lifetime.G_Status[GVL_Lifetime.G_Active_Device_Index].remaining_percent;
GVL_Lifetime.G_Active_Maintenance_Required := GVL_Lifetime.G_Status[GVL_Lifetime.G_Active_Device_Index].maintenance_required;
GVL_Lifetime.G_Active_Label := GVL_Lifetime.G_Device_Labels[GVL_Lifetime.G_Active_Device_Index];

// === LIFETIME HEALTH SUMMARY ===
GVL_Lifetime.G_Any_Maintenance_Required :=
    GVL_Lifetime.G_Status[1].maintenance_required OR
    GVL_Lifetime.G_Status[2].maintenance_required OR
    GVL_Lifetime.G_Status[3].maintenance_required OR
    GVL_Lifetime.G_Status[4].maintenance_required;

GVL_Lifetime.G_Maintenance_Warning :=
    (GVL_Lifetime.G_Status[1].remaining_percent <= 20) OR
    (GVL_Lifetime.G_Status[2].remaining_percent <= 20) OR
    (GVL_Lifetime.G_Status[3].remaining_percent <= 20) OR
    (GVL_Lifetime.G_Status[4].remaining_percent <= 20);

GVL_Lifetime.G_Maintenance_Critical :=
    (GVL_Lifetime.G_Status[1].remaining_percent <= 5) OR
    (GVL_Lifetime.G_Status[2].remaining_percent <= 5) OR
    (GVL_Lifetime.G_Status[3].remaining_percent <= 5) OR
    (GVL_Lifetime.G_Status[4].remaining_percent <= 5);

// === TREND → HISTORY WRITE (RATE-LIMITED SAFE MVP) ===
L_Trend_Write := (L_Trend_Data.record_count > 0);
L_Trend_Write_Allowed := FALSE;

IF L_Trend_Write AND NOT L_Trend_Write_Prev THEN
    IF (L_Trend_Last_Write_MS = 0) OR
       ((GVL_STATUS.G_System_Time_MS - L_Trend_Last_Write_MS) >= GVL_CONSTANTS.C_MS_IN_HOUR) THEN
        IF ABS(L_Trend_Avg - L_Trend_Last_Written_Avg) >= 0.5 THEN
            L_Trend_Write_Allowed := TRUE;
        END_IF;
    END_IF;

    IF L_Trend_Write_Allowed THEN
        L_Trend_Event.event_code := 1001;
        L_Trend_Event.event_value := L_Trend_Avg;
        L_Trend_Event.zone_id := 0;
        L_Trend_Event.operator_id := '';
        L_History_Write_Event := TRUE;
        L_History_Event := L_Trend_Event;

        L_Trend_Last_Write_MS := GVL_STATUS.G_System_Time_MS;
        L_Trend_Last_Written_Avg := L_Trend_Avg;
    END_IF;
END_IF;

L_Trend_Write_Prev := L_Trend_Write;

// >>> BULK_SYNC_ANCHOR: PRG_System <<<

// === EVENT LOGGING: FAULTS ===

// WATCHDOG
IF fbWatchdog.VO_Watchdog_Fault AND NOT L_Watchdog_Fault_Prev THEN
    fbLogEvent(
        VI_Event_Type := 11,
        VI_Timestamp := GVL_STATUS.G_System_Time_MS,
        VI_Param1 := 1,
        VI_Param2 := 1
    );
END_IF;

IF NOT fbWatchdog.VO_Watchdog_Fault AND L_Watchdog_Fault_Prev THEN
    fbLogEvent(
        VI_Event_Type := 12,
        VI_Timestamp := GVL_STATUS.G_System_Time_MS,
        VI_Param1 := 1,
        VI_Param2 := 0
    );
END_IF;

L_Watchdog_Fault_Prev := fbWatchdog.VO_Watchdog_Fault;

// IO
IF fbSystemHealth.VO_IO_Fault AND NOT L_IO_Fault_Prev THEN
    fbLogEvent(
        VI_Event_Type := 2,
        VI_Timestamp := GVL_STATUS.G_System_Time_MS,
        VI_Param1 := 1,
        VI_Param2 := 1
    );
END_IF;

IF NOT fbSystemHealth.VO_IO_Fault AND L_IO_Fault_Prev THEN
    fbLogEvent(
        VI_Event_Type := 3,
        VI_Timestamp := GVL_STATUS.G_System_Time_MS,
        VI_Param1 := 1,
        VI_Param2 := 0
    );
END_IF;

L_IO_Fault_Prev := fbSystemHealth.VO_IO_Fault;

// === EVENT LOGGING: MODE CHANGE ===
IF GVL_STATE.G_System_Mode <> L_Mode_Prev THEN
    fbLogEvent(
        VI_Event_Type := 4,
        VI_Timestamp := GVL_STATUS.G_System_Time_MS,
        VI_Param1 := TO_UDINT(L_Mode_Prev),
        VI_Param2 := TO_UDINT(GVL_STATE.G_System_Mode)
    );
END_IF;

L_Mode_Prev := GVL_STATE.G_System_Mode;

(* ---- PRG_System_Alarm_Gateway.st ---- *)
PROGRAM PRG_System_Alarm_Gateway
VAR
    fbSystemAlarmOrchestrator : FB_System_Alarm_Orchestrator;
    fbSystemGatewayIntent : FB_System_Gateway_Intent;
    L_Scenario_Req_Gateway : E_SCENARIO_TYPE;
END_VAR

// Default to no gateway scenario request each scan.
// The gateway FB may override it through the VIO parameter.
L_Scenario_Req_Gateway := SCENARIO_NONE;

fbSystemAlarmOrchestrator(
    VI_First_Fault_Active := GVL_SYSTEM_HEALTH.G_First_Fault_Active,
    VI_First_Fault_Type := GVL_SYSTEM_HEALTH.G_First_Fault_Type,
    VI_First_Fault_Source := GVL_SYSTEM_HEALTH.G_First_Fault_Source
);

fbSystemGatewayIntent(
    VI_System_Time_MS := GVL_TIME_SERVICE.G_Now_MS,
    VI_IsActivePLC := GVL_STATUS.G_Is_Active_PLC,
    VI_Gateway_Writes_Allowed := NOT GVL_STATUS.G_Diagnostics.Operator_Action_Blocked,
    VIO_FloorHeating_Temps := GVL_STATE.G_Floor_Temps,
    VIO_Zone_Valve_States := GVL_STATE.G_Zone_Valves,
    VIO_Lighting_Base_Levels := GVL_STATE.G_Lighting_Levels,
    VIO_Scenario_Req_Gateway := L_Scenario_Req_Gateway
);

GVL_INTENT_USER.I_Scenario_Request := L_Scenario_Req_Gateway;

END_PROGRAM

(* ---- PRG_System_BlackBox.st ---- *)
PROGRAM PRG_System_BlackBox
VAR
    fbBlackBox : FB_BlackBox_Recorder;
    L_BB_Record : ST_BlackBox_Record;
    L_BB_Freeze : BOOL;
    L_BB_Gas_Active : BOOL;
    L_BB_Fire_Active : BOOL;
    L_BB_Flood_Active : BOOL;
END_VAR

// BlackBox must record authoritative safety truth and latches,
// not stale alarm projection fields.
L_BB_Gas_Active := GVL_HEALTH_BRIDGE.G_Gas_Detected OR GVL_HEALTH_BRIDGE.G_CO_Alarm_Level OR GVL_STATE.G_Safety_Gas_Latched;
L_BB_Fire_Active := GVL_HEALTH_BRIDGE.G_Smoke_Detected OR GVL_STATE.G_Safety_Smoke_Latched;
L_BB_Flood_Active := GVL_HEALTH_BRIDGE.G_Leak_Detected OR GVL_STATE.G_Safety_Leak_Latched;

L_BB_Record.Timestamp := GVL_TIME_SERVICE.G_Now_MS;
L_BB_Record.PLC_Active_ID := GVL_STATUS.G_PLC_ID;
L_BB_Record.Gas_Methane_LEL := GVL_STATE.G_Methane_Sensors[1];
L_BB_Record.Gas_CO_PPM := GVL_STATE.G_CO_Sensors[1];
L_BB_Record.Flood_Active := L_BB_Flood_Active;
L_BB_Record.Fire_Active := L_BB_Fire_Active;

L_BB_Record.System_Mode := TO_BYTE(TO_INT(GVL_STATE.G_System_Mode));
L_BB_Record.First_Fault_Type := TO_BYTE(GVL_SYSTEM_HEALTH.G_First_Fault_Type);
L_BB_Record.First_Fault_Source := TO_BYTE(GVL_SYSTEM_HEALTH.G_First_Fault_Source);
L_BB_Record.First_Fault_Active := GVL_SYSTEM_HEALTH.G_First_Fault_Active;
L_BB_Record.System_Severity := TO_BYTE(GVL_SYSTEM_HEALTH.G_System_Severity);
L_BB_Record.Root_Cause := TO_BYTE(GVL_SYSTEM_HEALTH.G_Root_Cause);
L_BB_Record.Watchdog_Fault := GVL_SYSTEM_HEALTH.G_Watchdog_Fault;

L_BB_Freeze := L_BB_Gas_Active OR L_BB_Fire_Active OR L_BB_Flood_Active OR GVL_SYSTEM_HEALTH.G_First_Fault_Active;

fbBlackBox(
    VI_Current_Data := L_BB_Record,
    VI_Freeze := L_BB_Freeze,
    VI_Reset := GVL_COMMAND.G_Reset_Errors
);

END_PROGRAM

(* ---- PRG_System_Coordinator.st ---- *)
PROGRAM PRG_System_Coordinator
VAR
    fbCoord : FB_System_Coordinator;
END_VAR

fbCoord(
    VI_Fire_Latched := GVL_STATE.G_Safety_Smoke_Latched,
    VI_Gas_Latched := GVL_STATE.G_Safety_Gas_Latched,
    VI_Leak_Latched := GVL_STATE.G_Safety_Leak_Latched,
    VI_IO_Degraded := NOT GVL_STATUS.G_IO_Modules_Online[1],
    VI_Ownership_Violation := GVL_TEST.G_Ownership_Violation,
    VI_Behavior_Mode := GVL_MODE.G_Current_Behavior_Mode
);

GVL_SYSTEM_COORDINATION.G_Block_Heating := fbCoord.VO_Block_Heating;
GVL_SYSTEM_COORDINATION.G_Block_Ventilation := fbCoord.VO_Block_Ventilation;
GVL_SYSTEM_COORDINATION.G_Block_Lighting_Override := fbCoord.VO_Block_Lighting;
GVL_SYSTEM_COORDINATION.G_Block_Sockets_Override := fbCoord.VO_Block_Sockets;

GVL_SYSTEM_COORDINATION.G_System_Degraded := fbCoord.VO_System_Degraded;
GVL_SYSTEM_COORDINATION.G_Coordination_Code := fbCoord.VO_Code;

(* ---- PRG_System_Diagnostics.st ---- *)
PROGRAM PRG_System_Diagnostics
VAR
    fbStateTraceLog : FB_State_Trace_Log;
    fbAdapt : FB_Behavior_Adapt;
    fbSystemDiagnosticsPublisher : FB_System_Diagnostics_Publisher;

    L_Pumps_4 : ARRAY[1..4] OF BOOL;
    L_Manifold_Pump_Out_Of_Service : ARRAY[1..GVL_CONSTANTS.C_MAX_MANIFOLDS] OF BOOL;
    L_Manifold_Pressure_Fault : ARRAY[1..GVL_CONSTANTS.C_MAX_MANIFOLDS] OF BOOL;
    L_Manifold_Current_Fault : ARRAY[1..GVL_CONSTANTS.C_MAX_MANIFOLDS] OF BOOL;
    L_Manifold_Return_Temp_Fault : ARRAY[1..GVL_CONSTANTS.C_MAX_MANIFOLDS] OF BOOL;
    L_i : INT;
    L_Last_State_Trace_MS : UDINT;

    L_Hum : REAL;
    L_PrevHum : REAL;
    L_DeltaHum : REAL;
    L_Confidence : REAL;
END_VAR

FOR L_i := 1 TO 4 DO
    L_Pumps_4[L_i] := GVL_HEATING_OUTPUT.DO_Manifold_Pumps[L_i];
END_FOR;

FOR L_i := 1 TO GVL_CONSTANTS.C_MAX_MANIFOLDS DO
    L_Manifold_Pump_Out_Of_Service[L_i] := NOT GVL_CONFIG.G_Manifold_Pump_In_Service[L_i];
    L_Manifold_Pressure_Fault[L_i] := GVL_HEATING_DIAGNOSTICS.G_Manifold_Pressure_Fault[L_i];
    L_Manifold_Current_Fault[L_i] := GVL_HEATING_DIAGNOSTICS.G_Manifold_Current_Fault[L_i];
    L_Manifold_Return_Temp_Fault[L_i] := GVL_HEATING_DIAGNOSTICS.G_Manifold_Return_Temp_Fault[L_i];
END_FOR;

fbStateTraceLog(
    VI_System_Time := GVL_TIME_SERVICE.G_Now_MS,
    VI_Gas_Alarm := GVL_HEALTH_BRIDGE.G_Gas_Detected OR GVL_HEALTH_BRIDGE.G_CO_Alarm_Level,
    VI_Leak_Alarm := GVL_HEALTH_BRIDGE.G_Leak_Detected,
    VI_Pumps := L_Pumps_4,
    VO_Last_Change_Time => L_Last_State_Trace_MS
);

FOR L_i := 1 TO GVL_CONSTANTS.C_MAX_ZONES DO

    L_Hum := GVL_INPUT.IN_Room_Hum[L_i];

    IF GVL_BEHAVIOR_ADAPT.G_Prev_Valid[L_i] THEN
        L_PrevHum := GVL_BEHAVIOR_ADAPT.G_Prev_Humidity[L_i];
    ELSE
        L_PrevHum := L_Hum;
    END_IF;

    L_DeltaHum := L_PrevHum - L_Hum;

    IF ABS(L_DeltaHum) < 0.5 THEN
        L_Confidence := 0.2;
    ELSE
        L_Confidence := 1.0;
    END_IF;

    IF GVL_INTENT_BEHAVIOR.I_Request_Ventilation_Boost THEN
        fbAdapt(
            iScenario := REASON_SCENARIO_VENT_BOOST,
            iSuccess := (L_DeltaHum > 5.0),
            iMeasuredValue := L_Hum,
            iZone := L_i,
            iConfidence := L_Confidence
        );
    END_IF;

    GVL_BEHAVIOR_ADAPT.G_Prev_Humidity[L_i] := L_Hum;
    GVL_BEHAVIOR_ADAPT.G_Prev_Valid[L_i] := TRUE;

END_FOR;

IF GVL_INTENT_BEHAVIOR.I_Request_Night_Mode THEN
    fbAdapt(
        iScenario := REASON_SCENARIO_NIGHT,
        iSuccess := TRUE,
        iMeasuredValue := 0.0,
        iZone := 0,
        iConfidence := 1.0
    );
END_IF;

fbSystemDiagnosticsPublisher(
    VI_Enable := TRUE,
    VI_System_Time_MS := GVL_TIME_SERVICE.G_Now_MS,
    VI_Backup_Pump_Out_Of_Service := NOT GVL_CONFIG.G_Backup_Circulation_Pump_In_Service,
    VI_Electric_Heater_Out_Of_Service := NOT GVL_CONFIG.G_Electric_Heater_In_Service,
    VI_Manifold_Pump_Out_Of_Service := L_Manifold_Pump_Out_Of_Service,
    VI_DHW_Heating_Pump_Out_Of_Service := NOT GVL_CONFIG.G_DHW_Heating_Pump_In_Service,
    VI_DHW_Circ_Pump_Out_Of_Service := NOT GVL_CONFIG.G_DHW_Circ_Pump_In_Service,
    VI_User_Access_Level := GVL_COMMAND.CMD_User_Access_Level,
    VI_Dangerous_Action_Pending := GVL_COMMAND.CMD_Dangerous_Action_Request,
    VI_Dangerous_Action_Text := 'Dangerous action confirmation requested',
    VI_Sensor_Fault := GVL_STATE.G_Heating_Sensor_Fault OR GVL_STATE.G_DHW_Sensor_Fault,
    VI_IO_Offline := GVL_STATE.G_Heating_IO_Fault OR GVL_STATE.G_DHW_IO_Fault,
    VI_Subsystem_Degraded := GVL_STATE.G_Heating_Subsystem_Degraded OR GVL_STATE.G_DHW_Subsystem_Degraded,
    VI_Manifold_Pressure_Fault := L_Manifold_Pressure_Fault,
    VI_Manifold_Current_Fault := L_Manifold_Current_Fault,
    VI_Manifold_Return_Temp_Fault := L_Manifold_Return_Temp_Fault
);

GVL_System_Diagnostics_Publication.G_System_Diagnostics := fbSystemDiagnosticsPublisher.VO_Diagnostics;
GVL_System_Diagnostics_Publication.G_System_Diagnostics_Publication_Valid := fbSystemDiagnosticsPublisher.VO_Publication_Valid;
GVL_System_Diagnostics_Publication.G_System_Diagnostics_Status_Code := fbSystemDiagnosticsPublisher.VO_Status_Code;
GVL_System_Diagnostics_Publication.G_System_Diagnostics_Status_Text := fbSystemDiagnosticsPublisher.VO_Status_Text;

END_PROGRAM

(* ---- PRG_System_Diagnostics_Ext.st ---- *)
PROGRAM PRG_System_Diagnostics_Ext
VAR
    L_Error_Heating : BOOL;
    L_Error_Safety : BOOL;
    L_Error_IO : BOOL;
END_VAR

// --- Detect errors ---
L_Error_Heating := GVL_STATE.G_Heating_Subsystem_Degraded;
L_Error_Safety := GVL_STATE.G_Safety_Gas_Alarm OR GVL_STATE.G_Safety_Leak_Alarm OR GVL_STATE.G_Safety_Smoke_Alarm;
L_Error_IO := GVL_STATE.G_Heating_IO_Fault;

// --- Heating ---
IF L_Error_Heating THEN
    GVL_DIAGNOSTICS_EXT.G_Error_Count_Heating := GVL_DIAGNOSTICS_EXT.G_Error_Count_Heating + 1;
    GVL_DIAGNOSTICS_EXT.G_Last_Error_Time_Heating := GVL_TIME_SERVICE.G_Now_MS;
    GVL_DIAGNOSTICS_EXT.G_Health_Heating := GVL_DIAGNOSTICS_EXT.G_Health_Heating - 0.05;
ELSE
    GVL_DIAGNOSTICS_EXT.G_Health_Heating := GVL_DIAGNOSTICS_EXT.G_Health_Heating + 0.01;
END_IF;

// Clamp
IF GVL_DIAGNOSTICS_EXT.G_Health_Heating < 0.0 THEN
    GVL_DIAGNOSTICS_EXT.G_Health_Heating := 0.0;
ELSIF GVL_DIAGNOSTICS_EXT.G_Health_Heating > 1.0 THEN
    GVL_DIAGNOSTICS_EXT.G_Health_Heating := 1.0;
END_IF;

// --- Safety ---
IF L_Error_Safety THEN
    GVL_DIAGNOSTICS_EXT.G_Error_Count_Safety := GVL_DIAGNOSTICS_EXT.G_Error_Count_Safety + 1;
    GVL_DIAGNOSTICS_EXT.G_Last_Error_Time_Safety := GVL_TIME_SERVICE.G_Now_MS;
    GVL_DIAGNOSTICS_EXT.G_Health_Safety := GVL_DIAGNOSTICS_EXT.G_Health_Safety - 0.1;
ELSE
    GVL_DIAGNOSTICS_EXT.G_Health_Safety := GVL_DIAGNOSTICS_EXT.G_Health_Safety + 0.02;
END_IF;

IF GVL_DIAGNOSTICS_EXT.G_Health_Safety < 0.0 THEN
    GVL_DIAGNOSTICS_EXT.G_Health_Safety := 0.0;
ELSIF GVL_DIAGNOSTICS_EXT.G_Health_Safety > 1.0 THEN
    GVL_DIAGNOSTICS_EXT.G_Health_Safety := 1.0;
END_IF;

// --- IO ---
IF L_Error_IO THEN
    GVL_DIAGNOSTICS_EXT.G_Error_Count_IO := GVL_DIAGNOSTICS_EXT.G_Error_Count_IO + 1;
    GVL_DIAGNOSTICS_EXT.G_Last_Error_Time_IO := GVL_TIME_SERVICE.G_Now_MS;
    GVL_DIAGNOSTICS_EXT.G_Health_IO := GVL_DIAGNOSTICS_EXT.G_Health_IO - 0.05;
ELSE
    GVL_DIAGNOSTICS_EXT.G_Health_IO := GVL_DIAGNOSTICS_EXT.G_Health_IO + 0.01;
END_IF;

IF GVL_DIAGNOSTICS_EXT.G_Health_IO < 0.0 THEN
    GVL_DIAGNOSTICS_EXT.G_Health_IO := 0.0;
ELSIF GVL_DIAGNOSTICS_EXT.G_Health_IO > 1.0 THEN
    GVL_DIAGNOSTICS_EXT.G_Health_IO := 1.0;
END_IF;

END_PROGRAM

(* ---- PRG_System_Health.st ---- *)
PROGRAM PRG_System_Health
VAR
    fbSystemHealthOrchestrator : FB_System_Health_Orchestrator;
END_VAR

// Centralized Health execution (Phase 5)
fbSystemHealthOrchestrator(
    VO_First_Fault_Active => GVL_SYSTEM_HEALTH.G_First_Fault_Active,
    VO_First_Fault_Type => GVL_SYSTEM_HEALTH.G_First_Fault_Type,
    VO_First_Fault_Source => GVL_SYSTEM_HEALTH.G_First_Fault_Source,
    VO_System_Severity => GVL_SYSTEM_HEALTH.G_System_Severity,
    VO_Root_Cause => GVL_SYSTEM_HEALTH.G_Root_Cause,
    VO_Watchdog_Fault => GVL_SYSTEM_HEALTH.G_Watchdog_Fault
);

END_PROGRAM

(* ---- PRG_System_History.st ---- *)
PROGRAM PRG_System_History
VAR
    fbHistoryManager : FB_History_Manager;
    L_History_Event : ST_History_Record;
    L_History_Write_Event : BOOL;
    L_Last_System_Mode : E_System_Operating_Mode;
    L_Last_Root_Cause : E_System_Root_Cause;
    L_Last_First_Fault_Source : INT;
    L_Last_Operator_Journal_Seq : UDINT;
    L_Last_Event_Code : UDINT;
    L_Last_Event_Value : REAL;
    L_Last_Event_Time_MS : UDINT;
END_VAR

L_History_Write_Event := FALSE;
L_History_Event.timestamp_ms := GVL_TIME_SERVICE.G_Now_MS;
L_History_Event.event_code := 0;
L_History_Event.event_value := 0.0;
L_History_Event.unit := 0;
L_History_Event.zone_id := 0;
L_History_Event.operator_id := 'SYSTEM';
L_History_Event.priority := E_ALERT_PRIORITY.ALERT_PRIORITY_HIGH;

IF GVL_STATE.G_System_Mode <> L_Last_System_Mode THEN
    L_History_Write_Event := TRUE;
    L_History_Event.event_code := 1101;
    L_History_Event.event_value := TO_REAL(TO_INT(GVL_STATE.G_System_Mode));
    L_History_Event.unit := 1;
    L_History_Event.zone_id := 0;
    L_History_Event.priority := E_ALERT_PRIORITY.ALERT_PRIORITY_HIGH;
    L_Last_System_Mode := GVL_STATE.G_System_Mode;

ELSIF GVL_SYSTEM_HEALTH.G_First_Fault_Active
      AND (GVL_SYSTEM_HEALTH.G_Root_Cause <> L_Last_Root_Cause) THEN
    L_History_Write_Event := TRUE;
    L_History_Event.event_code := 1102;
    L_History_Event.event_value := TO_REAL(TO_INT(GVL_SYSTEM_HEALTH.G_Root_Cause));
    L_History_Event.unit := 2;
    L_History_Event.zone_id := TO_BYTE(GVL_SYSTEM_HEALTH.G_First_Fault_Source);
    L_History_Event.priority := E_ALERT_PRIORITY.ALERT_PRIORITY_HIGH;
    L_Last_Root_Cause := GVL_SYSTEM_HEALTH.G_Root_Cause;

ELSIF GVL_SYSTEM_HEALTH.G_First_Fault_Active
      AND (GVL_SYSTEM_HEALTH.G_First_Fault_Source <> L_Last_First_Fault_Source) THEN
    L_History_Write_Event := TRUE;
    L_History_Event.event_code := 1103;
    L_History_Event.event_value := TO_REAL(GVL_SYSTEM_HEALTH.G_First_Fault_Source);
    L_History_Event.unit := 3;
    L_History_Event.zone_id := TO_BYTE(GVL_SYSTEM_HEALTH.G_First_Fault_Source);
    L_History_Event.priority := E_ALERT_PRIORITY.ALERT_PRIORITY_HIGH;
    L_Last_First_Fault_Source := GVL_SYSTEM_HEALTH.G_First_Fault_Source;

ELSIF GVL_STATUS.G_Current_Scenario <> GVL_STATUS.G_Previous_Scenario THEN
    L_History_Write_Event := TRUE;
    L_History_Event.event_code := 1001;
    L_History_Event.event_value := TO_REAL(GVL_STATUS.G_Current_Scenario);
    L_History_Event.unit := 4;
    L_History_Event.zone_id := 0;
    L_History_Event.priority := E_ALERT_PRIORITY.ALERT_PRIORITY_HIGH;
    GVL_STATUS.G_Previous_Scenario := GVL_STATUS.G_Current_Scenario;

ELSIF GVL_STATUS.G_Diagnostics.Alarm_Event_Pulse THEN
    L_History_Write_Event := TRUE;
    L_History_Event.event_code := GVL_STATUS.G_Diagnostics.Alarm_Event_Code;
    L_History_Event.event_value := GVL_STATUS.G_Diagnostics.Alarm_Event_Value;
    L_History_Event.unit := 10;
    L_History_Event.zone_id := 0;
    L_History_Event.priority := E_ALERT_PRIORITY.ALERT_PRIORITY_HIGH;

ELSIF GVL_STATUS.G_Diagnostics.Operator_Journal_Event_Seq <> L_Last_Operator_Journal_Seq THEN
    L_History_Write_Event := TRUE;
    L_History_Event.event_code := 1301;
    L_History_Event.event_value := TO_REAL(GVL_STATUS.G_Diagnostics.Operator_Journal_Event_Seq);
    L_History_Event.unit := 20;
    L_History_Event.zone_id := 0;
    L_History_Event.priority := E_ALERT_PRIORITY.ALERT_PRIORITY_HIGH;
    L_Last_Operator_Journal_Seq := GVL_STATUS.G_Diagnostics.Operator_Journal_Event_Seq;
END_IF;

IF NOT GVL_SYSTEM_HEALTH.G_First_Fault_Active THEN
    L_Last_Root_Cause := GVL_SYSTEM_HEALTH.G_Root_Cause;
    L_Last_First_Fault_Source := GVL_SYSTEM_HEALTH.G_First_Fault_Source;
END_IF;

IF L_History_Write_Event THEN
    IF (L_History_Event.event_code = L_Last_Event_Code)
       AND (ABS(L_History_Event.event_value - L_Last_Event_Value) < 0.001)
       AND (GVL_TIME_SERVICE.G_Now_MS - L_Last_Event_Time_MS < 5000) THEN
        L_History_Write_Event := FALSE;
    ELSE
        L_Last_Event_Code := L_History_Event.event_code;
        L_Last_Event_Value := L_History_Event.event_value;
        L_Last_Event_Time_MS := GVL_TIME_SERVICE.G_Now_MS;
    END_IF;
END_IF;

fbHistoryManager(
    VI_System_Time_MS := GVL_TIME_SERVICE.G_Now_MS,
    VI_Write_Event := L_History_Write_Event,
    VI_Event := L_History_Event
);

END_PROGRAM

(* ---- PRG_System_Init.st ---- *)
PROGRAM PRG_System_Init
VAR
    L_i : INT;
    L_Init_Done : BOOL := FALSE;
    L_Active_Zones_Count : INT;
    L_Zone_Index : INT;
END_VAR

IF L_Init_Done THEN
    RETURN;
END_IF;

L_Active_Zones_Count := GVL_SYSTEM_SIZE_CONFIG.G_Active_Heating_Circuits;

IF (L_Active_Zones_Count < 1) OR (L_Active_Zones_Count > GVL_CONSTANTS.C_MAX_HEATING_CIRCUITS) THEN
    GVL_STATUS.G_Diagnostics.Sensor_Fault := TRUE;
    GVL_STATUS.G_System_Mode_Text := 'CONFIG ERROR: invalid active heating circuits';
    GVL_COMMAND_SHADOW.G_Heating_Block := TRUE;
    GVL_COMMAND_SHADOW.G_Boiler_Stop := TRUE;
    L_Active_Zones_Count := GVL_CONSTANTS.C_MAX_HEATING_CIRCUITS;
END_IF;

FOR L_i := 1 TO L_Active_Zones_Count DO
    L_Zone_Index := GVL_CONFIG.G_Heating_Circuit_To_Zone[L_i];
    IF (L_Zone_Index < 1) OR (L_Zone_Index > GVL_CONSTANTS.C_MAX_ZONES) THEN
        GVL_STATUS.G_Diagnostics.Sensor_Fault := TRUE;
        GVL_STATUS.G_System_Mode_Text := CONCAT('CONFIG ERROR CIRCUIT ', INT_TO_STRING(L_i));
        GVL_COMMAND_SHADOW.G_Heating_Block := TRUE;
        GVL_COMMAND_SHADOW.G_Boiler_Stop := TRUE;
    END_IF;
END_FOR;

L_Init_Done := TRUE;

// >>> BULK_SYNC_ANCHOR: PRG_System_Init <<<

(* ---- PRG_System_Runtime_Base.st ---- *)
PROGRAM PRG_System_Runtime_Base
VAR
    fbSystemInit : FB_System_Init;
    fbSystemRecovery : FB_System_Recovery;
    fbSystemPersist : FB_System_Persist_Manager;
    fbSystemRedundancy : FB_System_Redundancy_Orchestrator;

    L_Local_State : ST_System_State_Snapshot;
    L_Remote_State : ST_System_State_Snapshot;

    L_Persist_Buffer : ARRAY[0..4] OF BYTE;
    L_Last_Written_Persist_Buffer : ARRAY[0..4] OF BYTE;
    L_Persist_Buffer_Changed : BOOL;
    L_Last_Persist_Write_MS : UDINT;
    L_Recovery_Done : BOOL;
    L_NVRAM_Cmd : BYTE;
    L_NVRAM_Offset : UDINT;
    L_NVRAM_Done : BOOL;
    L_NVRAM_Err : BOOL;
    L_NVRAM_ErrID : UDINT;
END_VAR

fbSystemInit(
    VIO_Local_State := L_Local_State,
    VIO_Remote_State := L_Remote_State
);

fbSystemRecovery(
    VIO_Recovery_Done := L_Recovery_Done
);

fbSystemPersist(
    VI_System_Time_MS := GVL_TIME_SERVICE.G_Now_MS,
    VI_IsActivePLC := GVL_STATUS.G_Is_Active_PLC,
    VIO_Persist_Buffer := L_Persist_Buffer,
    VIO_Last_Written_Persist_Buffer := L_Last_Written_Persist_Buffer,
    VIO_Persist_Buffer_Changed := L_Persist_Buffer_Changed,
    VIO_Last_Persist_Write_MS := L_Last_Persist_Write_MS,
    VIO_NVRAM_Cmd := L_NVRAM_Cmd,
    VIO_NVRAM_Offset := L_NVRAM_Offset,
    VIO_NVRAM_Done := L_NVRAM_Done,
    VIO_NVRAM_Err := L_NVRAM_Err,
    VIO_NVRAM_ErrID := L_NVRAM_ErrID
);

fbSystemRedundancy(
    VIO_Local_State := L_Local_State,
    VIO_Remote_State := L_Remote_State
);

END_PROGRAM

(* ---- PRG_System_Scenario_Rules.st ---- *)
PROGRAM PRG_System_Scenario_Rules
VAR
    fbSystemScenarioArb : FB_System_Scenario_Arbitration;
    fbRuleEngine : FB_Rule_Engine;
    L_i : INT;
    L_Scenario_Req_Operator : E_SCENARIO_TYPE;
    L_Scenario_Req_Gateway  : E_SCENARIO_TYPE;
    L_Scenario_Req_Rule     : E_SCENARIO_TYPE;
    L_Scenario_Req_Final    : E_SCENARIO_TYPE;
    L_Scenario_Intent       : E_SCENARIO_TYPE;
    L_Scenario_Source       : E_SCENARIO_SOURCE;

    // adapters
    L_Motion_16 : ARRAY[1..GVL_CONSTANTS.C_MAX_MANIFOLDS] OF BOOL;
END_VAR

// adapt motion sensors (32 → 16)
FOR L_i := 1 TO 16 DO
    L_Motion_16[L_i] := GVL_STATE.G_Motion_Sensors[L_i];
END_FOR;

IF GVL_STATE.G_System_Mode = E_System_Operating_Mode.MODE_NORMAL THEN
    L_Scenario_Req_Operator := GVL_COMMAND.G_Scenario_Request_Operator;
ELSE
    L_Scenario_Req_Operator := E_SCENARIO_TYPE.SCENARIO_NONE;
END_IF;

L_Scenario_Req_Gateway := GVL_INTENT_USER.I_Scenario_Request;
L_Scenario_Req_Rule := E_SCENARIO_TYPE.SCENARIO_NONE;

fbRuleEngine(
    VI_System_Time_MS := GVL_TIME_SERVICE.G_Now_MS,
    VI_IsActivePLC := GVL_STATUS.G_Is_Active_PLC,
    VI_Security_Armed := GVL_ALARM.G_Security_Armed,
    VI_Current_Time := GVL_TIME_SERVICE.G_Current_TOD,
    VI_Day_Of_Week := GVL_TIME_SERVICE.G_Day_Of_Week,
    VI_Rules := GVL_CONFIG.G_HMI_User_Rules,
    VI_Indoor_Temps := GVL_STATE.G_Room_Temps,
    VI_Floor_Temps := GVL_STATE.G_Floor_Temps,
    VI_Humidities := GVL_STATE.G_Room_Hum,
    VI_CO2_Levels := GVL_STATE.G_Room_CO2,
    VI_Motion_Sensors := L_Motion_16,
    VI_Door_Sensors := GVL_STATE.G_Door_Sensors,
    VI_Window_Sensors := GVL_STATE.G_Window_Sensors,
    VI_Water_Sensors := GVL_STATE.G_Water_Sensors,
    VI_Smoke_Sensors := GVL_STATE.G_Smoke_Sensors,
    VI_Methane_Sensors := GVL_STATE.G_Methane_Sensors,
    VI_CO_Sensors := GVL_STATE.G_CO_Sensors,
    VO_Actions => GVL_STATE.G_Rule_Actions
);

FOR L_i := 1 TO GVL_CONSTANTS.C_MAX_RULES DO
    IF GVL_STATE.G_Rule_Actions[L_i].Active AND GVL_STATE.G_Rule_Actions[L_i].Action_Type = E_Rule_Action_Type.ACTION_ACTIVATE_SCENARIO THEN
        L_Scenario_Req_Rule := TO_BYTE(GVL_STATE.G_Rule_Actions[L_i].Value);
    END_IF;
END_FOR;

fbSystemScenarioArb(
    VI_System_Time_MS := GVL_TIME_SERVICE.G_Now_MS,
    VI_IsActivePLC := GVL_STATUS.G_Is_Active_PLC,
    VI_System_Mode := GVL_STATE.G_System_Mode,
    VI_Security_Armed := GVL_ALARM.G_Security_Armed,
    VIO_Scenario_Req_Operator := L_Scenario_Req_Operator,
    VIO_Scenario_Req_Gateway := L_Scenario_Req_Gateway,
    VIO_Scenario_Req_Rule := L_Scenario_Req_Rule,
    VIO_Scenario_Req_Final := L_Scenario_Req_Final,
    VIO_Scenario_Intent := L_Scenario_Intent,
    VIO_Scenario_Source := L_Scenario_Source
);

END_PROGRAM

(* ---- PRG_System_Simulation.st ---- *)
PROGRAM PRG_System_Simulation
VAR
    fbSimulation : FB_Simulation_Manager;
    fbPlayback : FB_Presence_Playback;
    L_Playback_Lights : ARRAY[1..32] OF BOOL;
    L_Scenario_Config : ST_Scenario_Config;
END_VAR

L_Scenario_Config := GVL_CONFIG.G_HMI_Scenario_Configs[TO_INT(GVL_STATUS.G_Current_Scenario)];

fbSimulation(
    VI_System_Time_MS := GVL_TIME_SERVICE.G_Now_MS,
    VI_IsActivePLC := GVL_STATUS.G_Is_Active_PLC,
    VI_Scenario := GVL_STATUS.G_Current_Scenario,
    VI_Config := L_Scenario_Config
);

fbPlayback(
    VI_Mode_Record := FALSE,
    VI_Time_Index := GVL_TIME_SERVICE.G_Now_MS,
    VI_Light_Inputs := L_Playback_Lights
);

// Reset outputs
GVL_SIMULATION.G_Sim_Heating_Sensor_Fault := FALSE;
GVL_SIMULATION.G_Sim_IO_Fault := FALSE;
GVL_SIMULATION.G_Sim_Low_Pressure := FALSE;
GVL_SIMULATION.G_Sim_Predictive_Pump_Fault := FALSE;
GVL_SIMULATION.G_Sim_Gas_Alarm := FALSE;
GVL_SIMULATION.G_Sim_Leak_Alarm := FALSE;
GVL_SIMULATION.G_Sim_Smoke_Alarm := FALSE;
GVL_SIMULATION.G_Sim_Dual_PLC_Active := FALSE;

IF NOT GVL_SIMULATION.G_Simulation_Enable THEN
    GVL_SIMULATION.G_Test_Running := FALSE;
    GVL_SIMULATION.G_Test_Scenario_Active := FALSE;
    RETURN;
END_IF;

// Start scenario
IF GVL_SIMULATION.G_Test_Start THEN
    GVL_SIMULATION.G_Test_Scenario_Active := TRUE;
    GVL_SIMULATION.G_Test_Started_MS := GVL_TIME_SERVICE.G_Now_MS;
END_IF;

// Stop scenario
IF GVL_SIMULATION.G_Test_Stop THEN
    GVL_SIMULATION.G_Test_Scenario_Active := FALSE;
END_IF;

GVL_SIMULATION.G_Test_Running := GVL_SIMULATION.G_Test_Scenario_Active;

IF NOT GVL_SIMULATION.G_Test_Scenario_Active THEN
    RETURN;
END_IF;

// Scenario execution
CASE GVL_SIMULATION.G_Test_Scenario_ID OF

    1: // Gas safety
        GVL_SIMULATION.G_Sim_Gas_Alarm := TRUE;
        GVL_SIMULATION.G_Test_Expected_Result_Code := 1;

    2: // Leak + pressure
        GVL_SIMULATION.G_Sim_Leak_Alarm := TRUE;
        GVL_SIMULATION.G_Sim_Low_Pressure := TRUE;
        GVL_SIMULATION.G_Test_Expected_Result_Code := 2;

    3: // Sensor + predictive
        GVL_SIMULATION.G_Sim_Heating_Sensor_Fault := TRUE;
        GVL_SIMULATION.G_Sim_Predictive_Pump_Fault := TRUE;
        GVL_SIMULATION.G_Test_Expected_Result_Code := 2;

    4: // Dual PLC
        GVL_SIMULATION.G_Sim_Dual_PLC_Active := TRUE;
        GVL_SIMULATION.G_Test_Expected_Result_Code := 3;

    5: // Full stress
        GVL_SIMULATION.G_Sim_Gas_Alarm := TRUE;
        GVL_SIMULATION.G_Sim_Leak_Alarm := TRUE;
        GVL_SIMULATION.G_Sim_Smoke_Alarm := TRUE;
        GVL_SIMULATION.G_Sim_Low_Pressure := TRUE;
        GVL_SIMULATION.G_Sim_Predictive_Pump_Fault := TRUE;
        GVL_SIMULATION.G_Test_Expected_Result_Code := 4;

END_CASE;

// Auto stop by time
IF (GVL_TIME_SERVICE.G_Now_MS - GVL_SIMULATION.G_Test_Started_MS) > GVL_SIMULATION.G_Test_Duration_MS THEN
    GVL_SIMULATION.G_Test_Scenario_Active := FALSE;
END_IF;

END_PROGRAM
// >>> BULK_SYNC_ANCHOR: PRG_System_Simulation <<<

(* ---- PRG_System_Test_Harness.st ---- *)
PROGRAM PRG_System_Test_Harness
VAR
    L_i : INT;
    L_j : INT;
    L_Used : REAL;
    L_HP_Used : REAL;
    L_HP_Manifold_Adjusted : ARRAY[1..GVL_CONSTANTS.C_MAX_MANIFOLDS] OF INT;
    fbDecisionTest : FB_Heating_Decision_Context;
    fbDecisionHP : FB_Heating_Decision_Context;
    fbTestResult : FB_Test_Result_Handler;
    fbTrace : FB_Trace_Logger;
END_VAR

IF NOT GVL_TEST.G_Test_Enable THEN
    RETURN;
END_IF;

GVL_TEST.G_Test_Total_Checks := 0;
GVL_TEST.G_Test_Failed_Checks := 0;
GVL_TEST.G_Test_Passed := TRUE;
GVL_TEST.G_Test_Last_Failure_Index := 0;
GVL_TEST.G_Test_Last_Failure_Code := 0;

// Reset transient failure flags for this scan
GVL_TEST.G_Diagnostics_Duplicate_Event_Found := FALSE;
GVL_TEST.G_Diagnostics_Count_Out_Of_Range := FALSE;
GVL_TEST.G_Heating_Allocation_Budget_Exceeded := FALSE;
GVL_TEST.G_Heating_Allocation_Enabled_Not_Allowed := FALSE;
GVL_TEST.G_Safety_Latched_Without_Intent := FALSE;
GVL_TEST.G_HP_Adjusted_Priority_Lower_Bound_Violation := FALSE;
GVL_TEST.G_HP_Adjusted_Allocation_Budget_Exceeded := FALSE;
GVL_TEST.G_HP_Adjusted_Allocation_Enabled_Not_Allowed := FALSE;
GVL_TEST.G_HP_Guest_Preheat_Config_Out_Of_Range := FALSE;

// =========================
// TEST 1: Diagnostics count bounds
// =========================
GVL_TEST.G_Test_Total_Checks := GVL_TEST.G_Test_Total_Checks + 1;
IF (GVL_STATUS.G_Diagnostics_Count < 0) OR (GVL_STATUS.G_Diagnostics_Count > 50) THEN
    GVL_TEST.G_Diagnostics_Count_Out_Of_Range := TRUE;
    GVL_TEST.G_Test_Failed_Checks := GVL_TEST.G_Test_Failed_Checks + 1;
    GVL_TEST.G_Test_Passed := FALSE;
    GVL_TEST.G_Test_Last_Failure_Index := 1;
    GVL_TEST.G_Test_Last_Failure_Code := 1001;
END_IF;

// =========================
// TEST 2: Diagnostics duplicates
// =========================
GVL_TEST.G_Test_Total_Checks := GVL_TEST.G_Test_Total_Checks + 1;
FOR L_i := 1 TO GVL_STATUS.G_Diagnostics_Count DO
    FOR L_j := L_i + 1 TO GVL_STATUS.G_Diagnostics_Count DO
        IF (GVL_STATUS.G_Diagnostics_Events[L_i].Code = GVL_STATUS.G_Diagnostics_Events[L_j].Code) AND
           (GVL_STATUS.G_Diagnostics_Events[L_i].Source = GVL_STATUS.G_Diagnostics_Events[L_j].Source) THEN
            GVL_TEST.G_Diagnostics_Duplicate_Event_Found := TRUE;
            GVL_TEST.G_Test_Failed_Checks := GVL_TEST.G_Test_Failed_Checks + 1;
            GVL_TEST.G_Test_Passed := FALSE;
            GVL_TEST.G_Test_Last_Failure_Index := 2;
            GVL_TEST.G_Test_Last_Failure_Code := 1002;
        END_IF;
    END_FOR;
END_FOR;

// =========================
// TEST 3: Base heating decision consistency
// =========================
GVL_TEST.G_Test_Total_Checks := GVL_TEST.G_Test_Total_Checks + 1;
fbDecisionTest(
    VI_Manifold_Pump_In_Service := GVL_CONFIG.G_Manifold_Pump_In_Service,
    VI_Manifold_Pressure_Fault := GVL_STATUS.G_Diagnostics.Manifold_Pressure_Fault,
    VI_Manifold_Current_Fault := GVL_STATUS.G_Diagnostics.Manifold_Current_Fault,
    VI_Manifold_Thermal_Weight := GVL_CONFIG.G_Manifold_Thermal_Weight,
    VI_Manifold_Priority := GVL_CONFIG.G_Manifold_Priority,
    VI_Max_Thermal_Budget := GVL_CONFIG.G_Max_Thermal_Budget
);

L_Used := 0.0;
FOR L_i := 1 TO GVL_CONSTANTS.C_MAX_MANIFOLDS DO
    IF fbDecisionTest.VO_Manifold_Enabled[L_i] AND (NOT fbDecisionTest.VO_Manifold_Allowed[L_i]) THEN
        GVL_TEST.G_Heating_Allocation_Enabled_Not_Allowed := TRUE;
        GVL_TEST.G_Test_Failed_Checks := GVL_TEST.G_Test_Failed_Checks + 1;
        GVL_TEST.G_Test_Passed := FALSE;
        GVL_TEST.G_Test_Last_Failure_Index := 3;
        GVL_TEST.G_Test_Last_Failure_Code := 1003;
    END_IF;

    IF fbDecisionTest.VO_Manifold_Enabled[L_i] THEN
        L_Used := L_Used + GVL_CONFIG.G_Manifold_Thermal_Weight[L_i];
    END_IF;
END_FOR;

IF L_Used > (GVL_CONFIG.G_Max_Thermal_Budget + 0.001) THEN
    GVL_TEST.G_Heating_Allocation_Budget_Exceeded := TRUE;
    GVL_TEST.G_Test_Failed_Checks := GVL_TEST.G_Test_Failed_Checks + 1;
    GVL_TEST.G_Test_Passed := FALSE;
    GVL_TEST.G_Test_Last_Failure_Index := 3;
    GVL_TEST.G_Test_Last_Failure_Code := 1004;
END_IF;

// =========================
// TEST 4: Safety latch consistency
// =========================
GVL_TEST.G_Test_Total_Checks := GVL_TEST.G_Test_Total_Checks + 1;
IF GVL_STATE.G_Safety_Gas_Latched AND (NOT GVL_INTENT_SAFETY.I_Gas_Alarm_Active) THEN
    GVL_TEST.G_Safety_Latched_Without_Intent := TRUE;
    GVL_TEST.G_Test_Failed_Checks := GVL_TEST.G_Test_Failed_Checks + 1;
    GVL_TEST.G_Test_Passed := FALSE;
    GVL_TEST.G_Test_Last_Failure_Index := 4;
    GVL_TEST.G_Test_Last_Failure_Code := 1005;
END_IF;

// =========================
// TEST 5: HP policy adjusted priority
// =========================
GVL_TEST.G_Test_Total_Checks := GVL_TEST.G_Test_Total_Checks + 1;

IF (GVL_HEATING_POLICY_CONFIG.G_Guest_Preheat_Priority_Boost < 0) OR (GVL_HEATING_POLICY_CONFIG.G_Guest_Preheat_Priority_Boost > 10) THEN
    GVL_TEST.G_HP_Guest_Preheat_Config_Out_Of_Range := TRUE;
    GVL_TEST.G_Test_Failed_Checks := GVL_TEST.G_Test_Failed_Checks + 1;
    GVL_TEST.G_Test_Passed := FALSE;
    GVL_TEST.G_Test_Last_Failure_Index := 5;
    GVL_TEST.G_Test_Last_Failure_Code := 1007;
END_IF;

FOR L_i := 1 TO GVL_CONSTANTS.C_MAX_MANIFOLDS DO
    L_HP_Manifold_Adjusted[L_i] := GVL_CONFIG.G_Manifold_Priority[L_i];
END_FOR;

FOR L_i := 1 TO GVL_CONSTANTS.C_MAX_HEATING_CIRCUITS DO
    L_j := TO_INT(GVL_CONFIG.G_HMI_FloorHeating_Configs[L_i].manifold_id);

    IF (L_j >= 1) AND (L_j <= GVL_CONSTANTS.C_MAX_MANIFOLDS) THEN
        L_HP_Manifold_Adjusted[L_j] := L_HP_Manifold_Adjusted[L_j] + TO_INT(GVL_HEATING_POLICY.G_Zone_Priority_Bias[L_i]);

        IF GVL_HEATING_POLICY_CONFIG.G_Guest_Preheat_Enabled AND GVL_HEATING_POLICY.G_Zone_Guest_Preheat_Request[L_i] THEN
            L_HP_Manifold_Adjusted[L_j] := L_HP_Manifold_Adjusted[L_j] + GVL_HEATING_POLICY_CONFIG.G_Guest_Preheat_Priority_Boost;
        END_IF;

        IF L_HP_Manifold_Adjusted[L_j] < 1 THEN
            GVL_TEST.G_HP_Adjusted_Priority_Lower_Bound_Violation := TRUE;
            GVL_TEST.G_Test_Failed_Checks := GVL_TEST.G_Test_Failed_Checks + 1;
            GVL_TEST.G_Test_Passed := FALSE;
            GVL_TEST.G_Test_Last_Failure_Index := 5;
            GVL_TEST.G_Test_Last_Failure_Code := 1006;
        END_IF;
    END_IF;
END_FOR;

FOR L_i := 1 TO GVL_CONSTANTS.C_MAX_MANIFOLDS DO
    GVL_TEST.G_HP_Manifold_Adjusted_Priority[L_i] := L_HP_Manifold_Adjusted[L_i];
END_FOR;

fbDecisionHP(
    VI_Manifold_Pump_In_Service := GVL_CONFIG.G_Manifold_Pump_In_Service,
    VI_Manifold_Pressure_Fault := GVL_STATUS.G_Diagnostics.Manifold_Pressure_Fault,
    VI_Manifold_Current_Fault := GVL_STATUS.G_Diagnostics.Manifold_Current_Fault,
    VI_Manifold_Thermal_Weight := GVL_CONFIG.G_Manifold_Thermal_Weight,
    VI_Manifold_Priority := L_HP_Manifold_Adjusted,
    VI_Max_Thermal_Budget := GVL_CONFIG.G_Max_Thermal_Budget
);

L_HP_Used := 0.0;
FOR L_i := 1 TO GVL_CONSTANTS.C_MAX_MANIFOLDS DO
    IF fbDecisionHP.VO_Manifold_Enabled[L_i] AND (NOT fbDecisionHP.VO_Manifold_Allowed[L_i]) THEN
        GVL_TEST.G_HP_Adjusted_Allocation_Enabled_Not_Allowed := TRUE;
        GVL_TEST.G_Test_Failed_Checks := GVL_TEST.G_Test_Failed_Checks + 1;
        GVL_TEST.G_Test_Passed := FALSE;
        GVL_TEST.G_Test_Last_Failure_Index := 5;
        GVL_TEST.G_Test_Last_Failure_Code := 1008;
    END_IF;

    IF fbDecisionHP.VO_Manifold_Enabled[L_i] THEN
        L_HP_Used := L_HP_Used + GVL_CONFIG.G_Manifold_Thermal_Weight[L_i];
    END_IF;
END_FOR;

IF L_HP_Used > (GVL_CONFIG.G_Max_Thermal_Budget + 0.001) THEN
    GVL_TEST.G_HP_Adjusted_Allocation_Budget_Exceeded := TRUE;
    GVL_TEST.G_Test_Failed_Checks := GVL_TEST.G_Test_Failed_Checks + 1;
    GVL_TEST.G_Test_Passed := FALSE;
    GVL_TEST.G_Test_Last_Failure_Index := 5;
    GVL_TEST.G_Test_Last_Failure_Code := 1009;
END_IF;

IF GVL_TEST.G_Test_Passed THEN
    GVL_TEST.G_Test_Status_Msg := 'ALL TESTS PASSED';
ELSE
    GVL_TEST.G_Test_Status_Msg := 'TEST FAILURES DETECTED';
END_IF;

fbTestResult(
    VI_Test_Passed := GVL_TEST.G_Test_Passed
);

IF NOT GVL_TEST.G_Test_Passed THEN
    fbTrace(
        VI_Event_Code := UDINT_TO_INT(GVL_TEST.G_Test_Last_Failure_Code),
        VI_System_Time := GVL_STATUS.G_System_Time_MS
    );
END_IF;
END_PROGRAM

(* ---- PRG_System_Trend.st ---- *)
PROGRAM PRG_System_Trend
VAR
    fbTrendLogger : FB_Trend_Logger;
    L_TrendData : ST_Trend_Data;
END_VAR

// minimal trend: log room temperature 1
fbTrendLogger(
    VI_Value := GVL_STATE.G_Room_Temps[1],
    VIO_Trend_Data := L_TrendData
);

END_PROGRAM
